LIN {X 0,Y 249.026,Z 523.934,A -85,B 0,C 180,E1 -19032.796,E2 -19032.796} C_VEL
LIN {X 0,Y 250.402,Z 519.579,A -85,B 0,C 180,E1 -19035.438,E2 -19035.438} C_VEL
LIN {X 0,Y 252.113,Z 513.971,A -85,B 0,C 180,E1 -19038.007,E2 -19038.007} C_VEL
LIN {X 0,Y 254.478,Z 506.507,A -85,B 0,C 180,E1 -19040.637,E2 -19040.637} C_VEL
LIN {X 0,Y 257.002,Z 497.79,A -85,B 0,C 180,E1 -19043.014,E2 -19043.014} C_VEL
LIN {X 0,Y 259.635,Z 487.535,A -85,B 0,C 180,E1 -19045.223,E2 -19045.223} C_VEL
LIN {X 0,Y 262.011,Z 477.566,A -85,B 0,C 180,E1 -19046.899,E2 -19046.899} C_VEL
LIN {X 0,Y 264.202,Z 466.893,A -85,B 0,C 180,E1 -19048.33,E2 -19048.33} C_VEL
LIN {X 0,Y 266.285,Z 454.649,A -85,B 0,C 180,E1 -19049.606,E2 -19049.606} C_VEL
LIN {X 0,Y 267.921,Z 441.662,A -85,B 0,C 180,E1 -19050.602,E2 -19050.602} C_VEL
LIN {X 0,Y 269.029,Z 429.527,A -85,B 0,C 180,E1 -19051.238,E2 -19051.238} C_VEL
LIN {X 0,Y 270.232,Z 406.171,A -85,B 0,C 180,E1 -19051.957,E2 -19051.957} C_VEL
LIN {X 0,Y 272.221,Z 363.158,A -85,B 0,C 180,E1 -19053.174,E2 -19053.174} C_VEL
LIN {X 0,Y 265.544,Z 348.107,A -85,B 0,C 180,E1 -19054.833,E2 -19054.833} C_VEL
LIN {X 0,Y 258.825,Z 335.75,A -85,B 0,C 180,E1 -19056.552,E2 -19056.552} C_VEL
LIN {X 0,Y 254.137,Z 328.112,A -85,B 0,C 180,E1 -19057.811,E2 -19057.811} C_VEL
LIN {X 0,Y 251.084,Z 323.594,A -85,B 0,C 180,E1 -19058.661,E2 -19058.661} C_VEL
LIN {X 0,Y 249.464,Z 321.033,A -85,B 0,C 180,E1 -19059.136,E2 -19059.136} C_VEL
LIN {X 0,Y 249.221,Z 320.145,A -85,B 0,C 180,E1 -19059.29,E2 -19059.29} C_VEL
LIN {X 0,Y 249.065,Z 319.467,A -85,B 0,C 180,E1 -19059.777,E2 -19059.777} C_VEL
LIN {X 0,Y 249.159,Z 319.446,A -85,B 0,C 180,E1 -19063.616,E2 -19063.616} C_VEL
LIN {X 0,Y 249.193,Z 319.441,A -85,B 0,C 180,E1 -19068.614,E2 -19068.614} C_VEL
LIN {X 0,Y 249.408,Z 319.413,A -85,B 0,C 180,E1 -19071.9,E2 -19071.9} C_VEL
LIN {X 0,Y 249.252,Z 319.432,A -85,B 0,C 180,E1 -19075.148,E2 -19075.148} C_VEL
LIN {X 0,Y 249.36,Z 319.415,A -85,B 0,C 180,E1 -19076.547,E2 -19076.547} C_VEL
LIN {X 0,Y 249.147,Z 319.448,A -85,B 0,C 180,E1 -19077.45,E2 -19077.45} C_VEL
LIN {X 0,Y 247.894,Z 319.605,A -85,B 0,C 180,E1 -19078.785,E2 -19078.785} C_VEL
LIN {X 0,Y 242.676,Z 320.249,A -85,B 0,C 180,E1 -19082.817,E2 -19082.817} C_VEL
LIN {X 0,Y 242.282,Z 320.293,A -85,B 0,C 180,E1 -19083.759,E2 -19083.759} C_VEL
LIN {X 0,Y 242.387,Z 320.287,A -85,B 0,C 180,E1 -19086.66,E2 -19086.66} C_VEL
LIN {X 0,Y 242.274,Z 320.307,A -85,B 0,C 180,E1 -19090.023,E2 -19090.023} C_VEL
LIN {X 0,Y 242.104,Z 320.321,A -85,B 0,C 180,E1 -19095.145,E2 -19095.145} C_VEL
LIN {X 0,Y 242.049,Z 320.332,A -85,B 0,C 180,E1 -19098.626,E2 -19098.626} C_VEL
LIN {X 0,Y 242.035,Z 320.332,A -85,B 0,C 180,E1 -19102.178,E2 -19102.178} C_VEL
LIN {X 0,Y 242.033,Z 320.33,A -85,B 0,C 180,E1 -19105.842,E2 -19105.842} C_VEL
LIN {X 0,Y 241.997,Z 320.336,A -85,B 0,C 180,E1 -19109.585,E2 -19109.585} C_VEL
LIN {X 0,Y 241.961,Z 320.346,A -85,B 0,C 180,E1 -19113.496,E2 -19113.496} C_VEL
LIN {X 0,Y 242,Z 320.338,A -85,B 0,C 180,E1 -19117.58,E2 -19117.58} C_VEL
LIN {X 0,Y 242.017,Z 320.34,A -85,B 0,C 180,E1 -19121.906,E2 -19121.906} C_VEL
LIN {X 0,Y 242.019,Z 320.432,A -85,B 0,C 180,E1 -19125.685,E2 -19125.685} C_VEL
LIN {X 0,Y 244.031,Z 326.812,A -85,B 0,C 180,E1 -19129.112,E2 -19129.112} C_VEL
LIN {X 0,Y 245.742,Z 332.805,A -85,B 0,C 180,E1 -19132.023,E2 -19132.023} C_VEL
LIN {X 0,Y 248.529,Z 337.73,A -85,B 0,C 180,E1 -19132.878,E2 -19132.878} C_VEL
LIN {X 0,Y 254.858,Z 349.777,A -85,B 0,C 180,E1 -19134.724,E2 -19134.724} C_VEL
LIN {X 0,Y 260.505,Z 361.853,A -85,B 0,C 180,E1 -19136.281,E2 -19136.281} C_VEL
LIN {X 0,Y 262.541,Z 367.254,A -85,B 0,C 180,E1 -19136.855,E2 -19136.855} C_VEL
LIN {X 0,Y 264.938,Z 384.313,A -85,B 0,C 180,E1 -19137.905,E2 -19137.905} C_VEL
LIN {X 0,Y 265.403,Z 390.459,A -85,B 0,C 180,E1 -19138.206,E2 -19138.206} C_VEL
LIN {X 0,Y 262.759,Z 444.06,A -85,B 0,C 180,E1 -19139.798,E2 -19139.798} C_VEL
LIN {X 0,Y 261.252,Z 457.92,A -85,B 0,C 180,E1 -19140.495,E2 -19140.495} C_VEL
LIN {X 0,Y 259.436,Z 469.841,A -85,B 0,C 180,E1 -19141.378,E2 -19141.378} C_VEL
LIN {X 0,Y 257.137,Z 481.502,A -85,B 0,C 180,E1 -19142.542,E2 -19142.542} C_VEL
LIN {X 0,Y 254.668,Z 492.793,A -85,B 0,C 180,E1 -19144.025,E2 -19144.025} C_VEL
LIN {X 0,Y 252.027,Z 503.055,A -85,B 0,C 180,E1 -19145.72,E2 -19145.72} C_VEL
LIN {X 0,Y 249.478,Z 512.316,A -85,B 0,C 180,E1 -19147.655,E2 -19147.655} C_VEL
LIN {X 0,Y 246.894,Z 521.368,A -85,B 0,C 180,E1 -19150.033,E2 -19150.033} C_VEL
LIN {X 0,Y 244.72,Z 528.699,A -85,B 0,C 180,E1 -19152.457,E2 -19152.457} C_VEL
LIN {X 0,Y 242.867,Z 534.602,A -85,B 0,C 180,E1 -19154.911,E2 -19154.911} C_VEL
LIN {X 0,Y 241.478,Z 539.276,A -85,B 0,C 180,E1 -19157.398,E2 -19157.398} C_VEL
LIN {X 0,Y 240.6,Z 542.861,A -85,B 0,C 180,E1 -19159.912,E2 -19159.912} C_VEL
LIN {X 0,Y 240.202,Z 544.688,A -85,B 0,C 180,E1 -19161.594,E2 -19161.594} C_VEL
LIN {X 0,Y 239.799,Z 547.099,A -85,B 0,C 180,E1 -19164.962,E2 -19164.962} C_VEL
LIN {X 0,Y 239.799,Z 547.72,A -85,B 0,C 180,E1 -19166.645,E2 -19166.645} C_VEL
LIN {X 0,Y 239.903,Z 547.911,A -85,B 0,C 180,E1 -19168.327,E2 -19168.327} C_VEL
LIN {X 0,Y 239.958,Z 547.686,A -85,B 0,C 180,E1 -19170.005,E2 -19170.005} C_VEL
LIN {X 0,Y 239.917,Z 547.061,A -85,B 0,C 180,E1 -19171.684,E2 -19171.684} C_VEL
LIN {X 0,Y 239.841,Z 546.03,A -85,B 0,C 180,E1 -19173.365,E2 -19173.365} C_VEL
LIN {X 0,Y 239.849,Z 544.537,A -85,B 0,C 180,E1 -19175.048,E2 -19175.048} C_VEL
LIN {X 0,Y 240.047,Z 541.476,A -85,B 0,C 180,E1 -19177.576,E2 -19177.576} C_VEL
LIN {X 0,Y 240.503,Z 537.321,A -85,B 0,C 180,E1 -19180.103,E2 -19180.103} C_VEL
LIN {X 0,Y 241.444,Z 530.931,A -85,B 0,C 180,E1 -19183.042,E2 -19183.042} C_VEL
LIN {X 0,Y 242.804,Z 523.965,A -85,B 0,C 180,E1 -19185.535,E2 -19185.535} C_VEL
LIN {X 0,Y 244.46,Z 515.208,A -85,B 0,C 180,E1 -19188.006,E2 -19188.006} C_VEL
LIN {X 0,Y 246.228,Z 505.21,A -85,B 0,C 180,E1 -19190.252,E2 -19190.252} C_VEL
LIN {X 0,Y 248.095,Z 495.105,A -85,B 0,C 180,E1 -19192.05,E2 -19192.05} C_VEL
LIN {X 0,Y 249.963,Z 483.875,A -85,B 0,C 180,E1 -19193.623,E2 -19193.623} C_VEL
LIN {X 0,Y 251.793,Z 471.326,A -85,B 0,C 180,E1 -19194.975,E2 -19194.975} C_VEL
LIN {X 0,Y 253.237,Z 458.517,A -85,B 0,C 180,E1 -19195.978,E2 -19195.978} C_VEL
LIN {X 0,Y 254.374,Z 445.256,A -85,B 0,C 180,E1 -19196.674,E2 -19196.674} C_VEL
LIN {X 0,Y 256.515,Z 387.54,A -85,B 0,C 180,E1 -19198.405,E2 -19198.405} C_VEL
LIN {X 0,Y 252.725,Z 358.428,A -85,B 0,C 180,E1 -19199.754,E2 -19199.754} C_VEL
LIN {X 0,Y 251.517,Z 351.799,A -85,B 0,C 180,E1 -19200.103,E2 -19200.103} C_VEL
LIN {X 0,Y 245.361,Z 335.617,A -85,B 0,C 180,E1 -19201.356,E2 -19201.356} C_VEL
LIN {X 0,Y 243.532,Z 326.882,A -85,B 0,C 180,E1 -19204.762,E2 -19204.762} C_VEL
LIN {X 0,Y 242.052,Z 320.333,A -85,B 0,C 180,E1 -19207.459,E2 -19207.459} C_VEL
LIN {X 0,Y 241.941,Z 320.35,A -85,B 0,C 180,E1 -19211.925,E2 -19211.925} C_VEL
LIN {X 0,Y 241.933,Z 320.352,A -85,B 0,C 180,E1 -19216.575,E2 -19216.575} C_VEL
LIN {X 0,Y 242.001,Z 320.339,A -85,B 0,C 180,E1 -19221.642,E2 -19221.642} C_VEL
LIN {X 0,Y 241.986,Z 320.343,A -85,B 0,C 180,E1 -19224.489,E2 -19224.489} C_VEL
LIN {X 0,Y 241.975,Z 320.346,A -85,B 0,C 180,E1 -19228.48,E2 -19228.48} C_VEL
LIN {X 0,Y 242.006,Z 320.34,A -85,B 0,C 180,E1 -19232.312,E2 -19232.312} C_VEL
LIN {X 0,Y 242.044,Z 320.331,A -85,B 0,C 180,E1 -19236.015,E2 -19236.015} C_VEL
LIN {X 0,Y 241.998,Z 320.336,A -85,B 0,C 180,E1 -19239.604,E2 -19239.604} C_VEL
LIN {X 0,Y 242.12,Z 320.304,A -85,B 0,C 180,E1 -19243.319,E2 -19243.319} C_VEL
LIN {X 0,Y 242.168,Z 320.315,A -85,B 0,C 180,E1 -19248.279,E2 -19248.279} C_VEL
LIN {X 0,Y 242.399,Z 320.288,A -85,B 0,C 180,E1 -19251.665,E2 -19251.665} C_VEL
LIN {X 0,Y 242.423,Z 320.281,A -85,B 0,C 180,E1 -19253.341,E2 -19253.341} C_VEL
LIN {X 0,Y 242.636,Z 320.233,A -85,B 0,C 180,E1 -19258.34,E2 -19258.34} C_VEL
LIN {X 0,Y 242.634,Z 320.251,A -85,B 0,C 180,E1 -19261.66,E2 -19261.66} C_VEL
LIN {X 0,Y 242.395,Z 320.289,A -85,B 0,C 180,E1 -19266.66,E2 -19266.66} C_VEL
LIN {X 0,Y 242.266,Z 320.3,A -85,B 0,C 180,E1 -19270.024,E2 -19270.024} C_VEL
LIN {X 0,Y 242.126,Z 320.323,A -85,B 0,C 180,E1 -19275.144,E2 -19275.144} C_VEL
LIN {X 0,Y 242.026,Z 320.326,A -85,B 0,C 180,E1 -19278.628,E2 -19278.628} C_VEL
LIN {X 0,Y 241.978,Z 320.343,A -85,B 0,C 180,E1 -19282.183,E2 -19282.183} C_VEL
LIN {X 0,Y 241.992,Z 320.339,A -85,B 0,C 180,E1 -19285.826,E2 -19285.826} C_VEL
LIN {X 0,Y 241.967,Z 320.324,A -85,B 0,C 180,E1 -19289.589,E2 -19289.589} C_VEL
LIN {X 0,Y 241.973,Z 320.324,A -85,B 0,C 180,E1 -19293.494,E2 -19293.494} C_VEL
LIN {X 0,Y 241.971,Z 320.34,A -85,B 0,C 180,E1 -19297.585,E2 -19297.585} C_VEL
LIN {X 0,Y 241.905,Z 320.348,A -85,B 0,C 180,E1 -19301.93,E2 -19301.93} C_VEL
LIN {X 0,Y 241.891,Z 320.356,A -85,B 0,C 180,E1 -19306.582,E2 -19306.582} C_VEL
LIN {X 0,Y 241.936,Z 320.343,A -85,B 0,C 180,E1 -19310.273,E2 -19310.273} C_VEL
LIN {X 0,Y 241.981,Z 320.343,A -85,B 0,C 180,E1 -19314.484,E2 -19314.484} C_VEL
LIN {X 0,Y 241.937,Z 320.35,A -85,B 0,C 180,E1 -19318.47,E2 -19318.47} C_VEL
LIN {X 0,Y 241.968,Z 320.344,A -85,B 0,C 180,E1 -19322.304,E2 -19322.304} C_VEL
LIN {X 0,Y 242.03,Z 320.334,A -85,B 0,C 180,E1 -19326.009,E2 -19326.009} C_VEL
LIN {X 0,Y 242,Z 320.341,A -85,B 0,C 180,E1 -19329.6,E2 -19329.6} C_VEL
LIN {X 0,Y 242.122,Z 320.327,A -85,B 0,C 180,E1 -19333.312,E2 -19333.312} C_VEL
LIN {X 0,Y 242.173,Z 320.316,A -85,B 0,C 180,E1 -19338.274,E2 -19338.274} C_VEL
LIN {X 0,Y 242.376,Z 320.29,A -85,B 0,C 180,E1 -19341.659,E2 -19341.659} C_VEL
LIN {X 0,Y 242.4,Z 320.291,A -85,B 0,C 180,E1 -19343.335,E2 -19343.335} C_VEL
LIN {X 0,Y 242.622,Z 320.26,A -85,B 0,C 180,E1 -19348.335,E2 -19348.335} C_VEL
LIN {X 0,Y 242.638,Z 320.438,A -85,B 0,C 180,E1 -19350.461,E2 -19350.461} C_VEL
LIN {X 0,Y 243.698,Z 323.226,A -85,B 0,C 180,E1 -19350.686,E2 -19350.686} C_VEL
LIN {X 0,Y 247.603,Z 332.184,A -85,B 0,C 180,E1 -19351.45,E2 -19351.45} C_VEL
LIN {X 0,Y 254.32,Z 349.239,A -85,B 0,C 180,E1 -19352.752,E2 -19352.752} C_VEL
LIN {X 0,Y 257.363,Z 357.984,A -85,B 0,C 180,E1 -19353.352,E2 -19353.352} C_VEL
LIN {X 0,Y 254.717,Z 426.897,A -85,B 0,C 180,E1 -19355.391,E2 -19355.391} C_VEL
LIN {X 0,Y 253.733,Z 440.855,A -85,B 0,C 180,E1 -19356.14,E2 -19356.14} C_VEL
LIN {X 0,Y 252.489,Z 453.86,A -85,B 0,C 180,E1 -19357.19,E2 -19357.19} C_VEL
LIN {X 0,Y 250.977,Z 465.457,A -85,B 0,C 180,E1 -19358.448,E2 -19358.448} C_VEL
LIN {X 0,Y 249.262,Z 476.237,A -85,B 0,C 180,E1 -19359.939,E2 -19359.939} C_VEL
LIN {X 0,Y 247.528,Z 486.205,A -85,B 0,C 180,E1 -19361.665,E2 -19361.665} C_VEL
LIN {X 0,Y 245.738,Z 495.959,A -85,B 0,C 180,E1 -19363.791,E2 -19363.791} C_VEL
LIN {X 0,Y 243.947,Z 505.16,A -85,B 0,C 180,E1 -19366.307,E2 -19366.307} C_VEL
LIN {X 0,Y 242.666,Z 511.758,A -85,B 0,C 180,E1 -19368.57,E2 -19368.57} C_VEL
LIN {X 0,Y 241.472,Z 518.139,A -85,B 0,C 180,E1 -19371.352,E2 -19371.352} C_VEL
LIN {X 0,Y 240.693,Z 522.973,A -85,B 0,C 180,E1 -19374.121,E2 -19374.121} C_VEL
LIN {X 0,Y 240.213,Z 525.551,A -85,B 0,C 180,E1 -19376.023,E2 -19376.023} C_VEL
LIN {X 0,Y 239.738,Z 527.941,A -85,B 0,C 180,E1 -19378.422,E2 -19378.422} C_VEL
LIN {X 0,Y 239.585,Z 528.991,A -85,B 0,C 180,E1 -19379.904,E2 -19379.904} C_VEL
LIN {X 0,Y 239.562,Z 529.858,A -85,B 0,C 180,E1 -19381.866,E2 -19381.866} C_VEL
LIN {X 0,Y 239.738,Z 530.179,A -85,B 0,C 180,E1 -19384.832,E2 -19384.832} C_VEL
LIN {X 0,Y 240.236,Z 529.227,A -85,B 0,C 180,E1 -19387.894,E2 -19387.894} C_VEL
LIN {X 0,Y 241.105,Z 527.123,A -85,B 0,C 180,E1 -19390.722,E2 -19390.722} C_VEL
LIN {X 0,Y 242.246,Z 523.843,A -85,B 0,C 180,E1 -19393.506,E2 -19393.506} C_VEL
LIN {X 0,Y 243.754,Z 519.379,A -85,B 0,C 180,E1 -19396.213,E2 -19396.213} C_VEL
LIN {X 0,Y 245.683,Z 513.607,A -85,B 0,C 180,E1 -19398.857,E2 -19398.857} C_VEL
LIN {X 0,Y 248.116,Z 506.269,A -85,B 0,C 180,E1 -19401.452,E2 -19401.452} C_VEL
LIN {X 0,Y 250.841,Z 497.136,A -85,B 0,C 180,E1 -19403.958,E2 -19403.958} C_VEL
LIN {X 0,Y 253.34,Z 487.96,A -85,B 0,C 180,E1 -19405.958,E2 -19405.958} C_VEL
LIN {X 0,Y 255.802,Z 478.185,A -85,B 0,C 180,E1 -19407.65,E2 -19407.65} C_VEL
LIN {X 0,Y 258.155,Z 467.333,A -85,B 0,C 180,E1 -19409.136,E2 -19409.136} C_VEL
LIN {X 0,Y 260.397,Z 454.641,A -85,B 0,C 180,E1 -19410.483,E2 -19410.483} C_VEL
LIN {X 0,Y 262.048,Z 442.095,A -85,B 0,C 180,E1 -19411.458,E2 -19411.458} C_VEL
LIN {X 0,Y 263.222,Z 429.745,A -85,B 0,C 180,E1 -19412.116,E2 -19412.116} C_VEL
LIN {X 0,Y 264.502,Z 405.907,A -85,B 0,C 180,E1 -19412.86,E2 -19412.86} C_VEL
LIN {X 0,Y 266.484,Z 365.311,A -85,B 0,C 180,E1 -19414.027,E2 -19414.027} C_VEL
LIN {X 0,Y 260.565,Z 351.905,A -85,B 0,C 180,E1 -19415.587,E2 -19415.587} C_VEL
LIN {X 0,Y 254.402,Z 340.316,A -85,B 0,C 180,E1 -19417.247,E2 -19417.247} C_VEL
LIN {X 0,Y 249.596,Z 332.463,A -85,B 0,C 180,E1 -19418.604,E2 -19418.604} C_VEL
LIN {X 0,Y 247.303,Z 329.005,A -85,B 0,C 180,E1 -19419.274,E2 -19419.274} C_VEL
LIN {X 0,Y 245.279,Z 325.831,A -85,B 0,C 180,E1 -19419.889,E2 -19419.889} C_VEL
LIN {X 0,Y 242.726,Z 322.681,A -85,B 0,C 180,E1 -19420.66,E2 -19420.66} C_VEL
LIN {X 0,Y 242.084,Z 320.672,A -85,B 0,C 180,E1 -19420.937,E2 -19420.937} C_VEL
LIN {X 0,Y 242.029,Z 320.337,A -85,B 0,C 180,E1 -19421.372,E2 -19421.372} C_VEL
LIN {X 0,Y 242.102,Z 320.329,A -85,B 0,C 180,E1 -19424.855,E2 -19424.855} C_VEL
LIN {X 0,Y 242.275,Z 320.303,A -85,B 0,C 180,E1 -19430.443,E2 -19430.443} C_VEL
LIN {X 0,Y 242.379,Z 320.288,A -85,B 0,C 180,E1 -19433.34,E2 -19433.34} C_VEL
LIN {X 0,Y 242.594,Z 320.265,A -85,B 0,C 180,E1 -19438.34,E2 -19438.34} C_VEL
LIN {X 0,Y 242.594,Z 320.266,A -85,B 0,C 180,E1 -19441.66,E2 -19441.66} C_VEL
LIN {X 0,Y 242.282,Z 320.293,A -85,B 0,C 180,E1 -19443.759,E2 -19443.759} C_VEL
LIN {X 0,Y 241.536,Z 320.395,A -85,B 0,C 180,E1 -19445.148,E2 -19445.148} C_VEL
LIN {X 0,Y 238.687,Z 320.752,A -85,B 0,C 180,E1 -19447.415,E2 -19447.415} C_VEL
LIN {X 0,Y 235.469,Z 321.155,A -85,B 0,C 180,E1 -19450.211,E2 -19450.211} C_VEL
LIN {X 0,Y 235.112,Z 321.189,A -85,B 0,C 180,E1 -19451.179,E2 -19451.179} C_VEL
LIN {X 0,Y 235.058,Z 321.194,A -85,B 0,C 180,E1 -19455.61,E2 -19455.61} C_VEL
LIN {X 0,Y 234.994,Z 321.205,A -85,B 0,C 180,E1 -19459.207,E2 -19459.207} C_VEL
LIN {X 0,Y 234.963,Z 321.212,A -85,B 0,C 180,E1 -19462.883,E2 -19462.883} C_VEL
LIN {X 0,Y 234.936,Z 321.218,A -85,B 0,C 180,E1 -19466.662,E2 -19466.662} C_VEL
LIN {X 0,Y 234.899,Z 321.223,A -85,B 0,C 180,E1 -19470.572,E2 -19470.572} C_VEL
LIN {X 0,Y 234.931,Z 321.216,A -85,B 0,C 180,E1 -19474.638,E2 -19474.638} C_VEL
LIN {X 0,Y 234.971,Z 321.213,A -85,B 0,C 180,E1 -19478.967,E2 -19478.967} C_VEL
LIN {X 0,Y 234.972,Z 321.218,A -85,B 0,C 180,E1 -19483.467,E2 -19483.467} C_VEL
LIN {X 0,Y 234.962,Z 321.348,A -85,B 0,C 180,E1 -19484.064,E2 -19484.064} C_VEL
LIN {X 0,Y 237.368,Z 328.906,A -85,B 0,C 180,E1 -19488.388,E2 -19488.388} C_VEL
LIN {X 0,Y 238.399,Z 332.499,A -85,B 0,C 180,E1 -19490.185,E2 -19490.185} C_VEL
LIN {X 0,Y 241.186,Z 337.207,A -85,B 0,C 180,E1 -19491.131,E2 -19491.131} C_VEL
LIN {X 0,Y 245.517,Z 344.826,A -85,B 0,C 180,E1 -19492.512,E2 -19492.512} C_VEL
LIN {X 0,Y 251.337,Z 356.174,A -85,B 0,C 180,E1 -19494.275,E2 -19494.275} C_VEL
LIN {X 0,Y 257.128,Z 369.32,A -85,B 0,C 180,E1 -19495.947,E2 -19495.947} C_VEL
LIN {X 0,Y 259.348,Z 385.503,A -85,B 0,C 180,E1 -19496.986,E2 -19496.986} C_VEL
LIN {X 0,Y 259.804,Z 390.388,A -85,B 0,C 180,E1 -19497.255,E2 -19497.255} C_VEL
LIN {X 0,Y 257.015,Z 443.859,A -85,B 0,C 180,E1 -19498.878,E2 -19498.878} C_VEL
LIN {X 0,Y 255.445,Z 457.689,A -85,B 0,C 180,E1 -19499.583,E2 -19499.583} C_VEL
LIN {X 0,Y 253.465,Z 470.082,A -85,B 0,C 180,E1 -19500.525,E2 -19500.525} C_VEL
LIN {X 0,Y 250.919,Z 482.419,A -85,B 0,C 180,E1 -19501.802,E2 -19501.802} C_VEL
LIN {X 0,Y 248.352,Z 493.499,A -85,B 0,C 180,E1 -19503.313,E2 -19503.313} C_VEL
LIN {X 0,Y 245.597,Z 503.552,A -85,B 0,C 180,E1 -19505.041,E2 -19505.041} C_VEL
LIN {X 0,Y 242.946,Z 512.668,A -85,B 0,C 180,E1 -19507.02,E2 -19507.02} C_VEL
LIN {X 0,Y 240.217,Z 521.595,A -85,B 0,C 180,E1 -19509.454,E2 -19509.454} C_VEL
LIN {X 0,Y 237.933,Z 528.817,A -85,B 0,C 180,E1 -19511.939,E2 -19511.939} C_VEL
LIN {X 0,Y 235.986,Z 534.622,A -85,B 0,C 180,E1 -19514.46,E2 -19514.46} C_VEL
LIN {X 0,Y 234.519,Z 539.231,A -85,B 0,C 180,E1 -19517.018,E2 -19517.018} C_VEL
LIN {X 0,Y 233.572,Z 542.765,A -85,B 0,C 180,E1 -19519.606,E2 -19519.606} C_VEL
LIN {X 0,Y 233.17,Z 544.545,A -85,B 0,C 180,E1 -19521.338,E2 -19521.338} C_VEL
LIN {X 0,Y 232.728,Z 546.901,A -85,B 0,C 180,E1 -19524.808,E2 -19524.808} C_VEL
LIN {X 0,Y 232.704,Z 547.482,A -85,B 0,C 180,E1 -19526.543,E2 -19526.543} C_VEL
LIN {X 0,Y 232.81,Z 547.63,A -85,B 0,C 180,E1 -19528.276,E2 -19528.276} C_VEL
LIN {X 0,Y 232.888,Z 547.38,A -85,B 0,C 180,E1 -19530.006,E2 -19530.006} C_VEL
LIN {X 0,Y 232.825,Z 546.728,A -85,B 0,C 180,E1 -19531.735,E2 -19531.735} C_VEL
LIN {X 0,Y 232.767,Z 544.462,A -85,B 0,C 180,E1 -19534.875,E2 -19534.875} C_VEL
LIN {X 0,Y 233.001,Z 541.005,A -85,B 0,C 180,E1 -19537.806,E2 -19537.806} C_VEL
LIN {X 0,Y 233.482,Z 536.786,A -85,B 0,C 180,E1 -19540.41,E2 -19540.41} C_VEL
LIN {X 0,Y 234.502,Z 530.329,A -85,B 0,C 180,E1 -19543.435,E2 -19543.435} C_VEL
LIN {X 0,Y 235.887,Z 523.268,A -85,B 0,C 180,E1 -19546.002,E2 -19546.002} C_VEL
LIN {X 0,Y 237.533,Z 514.944,A -85,B 0,C 180,E1 -19548.4,E2 -19548.4} C_VEL
LIN {X 0,Y 239.343,Z 505.269,A -85,B 0,C 180,E1 -19550.636,E2 -19550.636} C_VEL
LIN {X 0,Y 241.259,Z 495.249,A -85,B 0,C 180,E1 -19552.483,E2 -19552.483} C_VEL
LIN {X 0,Y 243.177,Z 484.12,A -85,B 0,C 180,E1 -19554.097,E2 -19554.097} C_VEL
LIN {X 0,Y 245.041,Z 471.695,A -85,B 0,C 180,E1 -19555.485,E2 -19555.485} C_VEL
LIN {X 0,Y 246.505,Z 459.954,A -85,B 0,C 180,E1 -19556.458,E2 -19556.458} C_VEL
LIN {X 0,Y 247.657,Z 446.77,A -85,B 0,C 180,E1 -19557.21,E2 -19557.21} C_VEL
LIN {X 0,Y 248.591,Z 425.841,A -85,B 0,C 180,E1 -19557.908,E2 -19557.908} C_VEL
LIN {X 0,Y 249.931,Z 387.258,A -85,B 0,C 180,E1 -19559.071,E2 -19559.071} C_VEL
LIN {X 0,Y 245.978,Z 357.308,A -85,B 0,C 180,E1 -19560.508,E2 -19560.508} C_VEL
LIN {X 0,Y 245.065,Z 353.574,A -85,B 0,C 180,E1 -19560.739,E2 -19560.739} C_VEL
LIN {X 0,Y 238.12,Z 335.305,A -85,B 0,C 180,E1 -19562.234,E2 -19562.234} C_VEL
LIN {X 0,Y 235.775,Z 324.601,A -85,B 0,C 180,E1 -19566.599,E2 -19566.599} C_VEL
LIN {X 0,Y 234.96,Z 321.22,A -85,B 0,C 180,E1 -19568.096,E2 -19568.096} C_VEL
LIN {X 0,Y 234.888,Z 321.231,A -85,B 0,C 180,E1 -19571.581,E2 -19571.581} C_VEL
LIN {X 0,Y 234.891,Z 321.229,A -85,B 0,C 180,E1 -19575.9,E2 -19575.9} C_VEL
LIN {X 0,Y 234.88,Z 321.227,A -85,B 0,C 180,E1 -19578.831,E2 -19578.831} C_VEL
LIN {X 0,Y 234.923,Z 321.222,A -85,B 0,C 180,E1 -19583.25,E2 -19583.25} C_VEL
LIN {X 0,Y 234.96,Z 321.218,A -85,B 0,C 180,E1 -19587.425,E2 -19587.425} C_VEL
LIN {X 0,Y 234.942,Z 321.22,A -85,B 0,C 180,E1 -19591.405,E2 -19591.405} C_VEL
LIN {X 0,Y 234.983,Z 321.212,A -85,B 0,C 180,E1 -19595.246,E2 -19595.246} C_VEL
LIN {X 0,Y 234.95,Z 321.218,A -85,B 0,C 180,E1 -19598.964,E2 -19598.964} C_VEL
LIN {X 0,Y 235.062,Z 321.183,A -85,B 0,C 180,E1 -19603.094,E2 -19603.094} C_VEL
LIN {X 0,Y 235.1,Z 321.196,A -85,B 0,C 180,E1 -19607.921,E2 -19607.921} C_VEL
LIN {X 0,Y 235.328,Z 321.17,A -85,B 0,C 180,E1 -19611.412,E2 -19611.412} C_VEL
LIN {X 0,Y 235.373,Z 321.161,A -85,B 0,C 180,E1 -19613.14,E2 -19613.14} C_VEL
LIN {X 0,Y 235.595,Z 321.108,A -85,B 0,C 180,E1 -19618.291,E2 -19618.291} C_VEL
LIN {X 0,Y 235.594,Z 321.128,A -85,B 0,C 180,E1 -19621.709,E2 -19621.709} C_VEL
LIN {X 0,Y 235.345,Z 321.167,A -85,B 0,C 180,E1 -19626.86,E2 -19626.86} C_VEL
LIN {X 0,Y 235.191,Z 321.18,A -85,B 0,C 180,E1 -19630.329,E2 -19630.329} C_VEL
LIN {X 0,Y 235.075,Z 321.203,A -85,B 0,C 180,E1 -19635.609,E2 -19635.609} C_VEL
LIN {X 0,Y 234.967,Z 321.205,A -85,B 0,C 180,E1 -19639.209,E2 -19639.209} C_VEL
LIN {X 0,Y 234.921,Z 321.219,A -85,B 0,C 180,E1 -19642.887,E2 -19642.887} C_VEL
LIN {X 0,Y 234.91,Z 321.214,A -85,B 0,C 180,E1 -19646.665,E2 -19646.665} C_VEL
LIN {X 0,Y 234.891,Z 321.193,A -85,B 0,C 180,E1 -19650.574,E2 -19650.574} C_VEL
LIN {X 0,Y 234.905,Z 321.212,A -85,B 0,C 180,E1 -19654.643,E2 -19654.643} C_VEL
LIN {X 0,Y 234.92,Z 321.221,A -85,B 0,C 180,E1 -19658.934,E2 -19658.934} C_VEL
LIN {X 0,Y 234.86,Z 321.225,A -85,B 0,C 180,E1 -19664.092,E2 -19664.092} C_VEL
LIN {X 0,Y 234.852,Z 321.226,A -85,B 0,C 180,E1 -19668.821,E2 -19668.821} C_VEL
LIN {X 0,Y 234.926,Z 321.222,A -85,B 0,C 180,E1 -19671.076,E2 -19671.076} C_VEL
LIN {X 0,Y 234.905,Z 321.22,A -85,B 0,C 180,E1 -19675.354,E2 -19675.354} C_VEL
LIN {X 0,Y 234.894,Z 321.226,A -85,B 0,C 180,E1 -19679.423,E2 -19679.423} C_VEL
LIN {X 0,Y 234.976,Z 321.217,A -85,B 0,C 180,E1 -19683.804,E2 -19683.804} C_VEL
LIN {X 0,Y 234.973,Z 321.218,A -85,B 0,C 180,E1 -19688.004,E2 -19688.004} C_VEL
LIN {X 0,Y 235.063,Z 321.209,A -85,B 0,C 180,E1 -19693.088,E2 -19693.088} C_VEL
LIN {X 0,Y 235.104,Z 321.197,A -85,B 0,C 180,E1 -19697.917,E2 -19697.917} C_VEL
LIN {X 0,Y 235.316,Z 321.169,A -85,B 0,C 180,E1 -19701.407,E2 -19701.407} C_VEL
LIN {X 0,Y 235.352,Z 321.168,A -85,B 0,C 180,E1 -19703.135,E2 -19703.135} C_VEL
LIN {X 0,Y 235.58,Z 321.137,A -85,B 0,C 180,E1 -19708.285,E2 -19708.285} C_VEL
LIN {X 0,Y 235.584,Z 321.142,A -85,B 0,C 180,E1 -19709.621,E2 -19709.621} C_VEL
LIN {X 0,Y 236.502,Z 323.833,A -85,B 0,C 180,E1 -19709.835,E2 -19709.835} C_VEL
LIN {X 0,Y 240.954,Z 333.301,A -85,B 0,C 180,E1 -19710.72,E2 -19710.72} C_VEL
LIN {X 0,Y 248.512,Z 352.797,A -85,B 0,C 180,E1 -19712.259,E2 -19712.259} C_VEL
LIN {X 0,Y 250.863,Z 360.046,A -85,B 0,C 180,E1 -19712.754,E2 -19712.754} C_VEL
LIN {X 0,Y 248.133,Z 427.294,A -85,B 0,C 180,E1 -19714.792,E2 -19714.792} C_VEL
LIN {X 0,Y 247.136,Z 440.947,A -85,B 0,C 180,E1 -19715.542,E2 -19715.542} C_VEL
LIN {X 0,Y 245.909,Z 453.423,A -85,B 0,C 180,E1 -19716.559,E2 -19716.559} C_VEL
LIN {X 0,Y 244.353,Z 465.146,A -85,B 0,C 180,E1 -19717.846,E2 -19717.846} C_VEL
LIN {X 0,Y 242.514,Z 476.378,A -85,B 0,C 180,E1 -19719.428,E2 -19719.428} C_VEL
LIN {X 0,Y 240.533,Z 487.213,A -85,B 0,C 180,E1 -19721.368,E2 -19721.368} C_VEL
LIN {X 0,Y 238.674,Z 497.228,A -85,B 0,C 180,E1 -19723.658,E2 -19723.658} C_VEL
LIN {X 0,Y 237.028,Z 505.179,A -85,B 0,C 180,E1 -19725.911,E2 -19725.911} C_VEL
LIN {X 0,Y 235.658,Z 512.068,A -85,B 0,C 180,E1 -19728.333,E2 -19728.333} C_VEL
LIN {X 0,Y 234.454,Z 518.205,A -85,B 0,C 180,E1 -19731.075,E2 -19731.075} C_VEL
LIN {X 0,Y 233.651,Z 523.118,A -85,B 0,C 180,E1 -19733.95,E2 -19733.95} C_VEL
LIN {X 0,Y 232.895,Z 526.79,A -85,B 0,C 180,E1 -19736.906,E2 -19736.906} C_VEL
LIN {X 0,Y 232.597,Z 528.531,A -85,B 0,C 180,E1 -19738.902,E2 -19738.902} C_VEL
LIN {X 0,Y 232.461,Z 530.174,A -85,B 0,C 180,E1 -19742.164,E2 -19742.164} C_VEL
LIN {X 0,Y 232.692,Z 530.432,A -85,B 0,C 180,E1 -19745.365,E2 -19745.365} C_VEL
LIN {X 0,Y 233.279,Z 529.383,A -85,B 0,C 180,E1 -19748.436,E2 -19748.436} C_VEL
LIN {X 0,Y 234.251,Z 527.123,A -85,B 0,C 180,E1 -19751.405,E2 -19751.405} C_VEL
LIN {X 0,Y 235.499,Z 523.75,A -85,B 0,C 180,E1 -19754.255,E2 -19754.255} C_VEL
LIN {X 0,Y 237.162,Z 519.183,A -85,B 0,C 180,E1 -19757.033,E2 -19757.033} C_VEL
LIN {X 0,Y 239.3,Z 513.24,A -85,B 0,C 180,E1 -19759.769,E2 -19759.769} C_VEL
LIN {X 0,Y 241.874,Z 505.792,A -85,B 0,C 180,E1 -19762.397,E2 -19762.397} C_VEL
LIN {X 0,Y 244.481,Z 497.537,A -85,B 0,C 180,E1 -19764.695,E2 -19764.695} C_VEL
LIN {X 0,Y 247.022,Z 488.674,A -85,B 0,C 180,E1 -19766.678,E2 -19766.678} C_VEL
LIN {X 0,Y 249.581,Z 479.074,A -85,B 0,C 180,E1 -19768.393,E2 -19768.393} C_VEL
LIN {X 0,Y 252.243,Z 467.298,A -85,B 0,C 180,E1 -19770.042,E2 -19770.042} C_VEL
LIN {X 0,Y 254.524,Z 454.918,A -85,B 0,C 180,E1 -19771.372,E2 -19771.372} C_VEL
LIN {X 0,Y 256.266,Z 442.397,A -85,B 0,C 180,E1 -19772.361,E2 -19772.361} C_VEL
LIN {X 0,Y 257.444,Z 430.603,A -85,B 0,C 180,E1 -19773.01,E2 -19773.01} C_VEL
LIN {X 0,Y 258.615,Z 410.729,A -85,B 0,C 180,E1 -19773.662,E2 -19773.662} C_VEL
LIN {X 0,Y 260.787,Z 367.352,A -85,B 0,C 180,E1 -19774.947,E2 -19774.947} C_VEL
LIN {X 0,Y 255.671,Z 355.747,A -85,B 0,C 180,E1 -19776.361,E2 -19776.361} C_VEL
LIN {X 0,Y 249.838,Z 344.615,A -85,B 0,C 180,E1 -19778.026,E2 -19778.026} C_VEL
LIN {X 0,Y 244.951,Z 336.58,A -85,B 0,C 180,E1 -19779.477,E2 -19779.477} C_VEL
LIN {X 0,Y 240.811,Z 330.383,A -85,B 0,C 180,E1 -19780.777,E2 -19780.777} C_VEL
LIN {X 0,Y 238.564,Z 327.157,A -85,B 0,C 180,E1 -19781.52,E2 -19781.52} C_VEL
LIN {X 0,Y 238,Z 326.175,A -85,B 0,C 180,E1 -19781.72,E2 -19781.72} C_VEL
LIN {X 0,Y 235.951,Z 323.972,A -85,B 0,C 180,E1 -19782.39,E2 -19782.39} C_VEL
LIN {X 0,Y 235.038,Z 321.21,A -85,B 0,C 180,E1 -19782.823,E2 -19782.823} C_VEL
LIN {X 0,Y 235.043,Z 321.203,A -85,B 0,C 180,E1 -19786.16,E2 -19786.16} C_VEL
LIN {X 0,Y 235.283,Z 321.177,A -85,B 0,C 180,E1 -19791.411,E2 -19791.411} C_VEL
LIN {X 0,Y 235.329,Z 321.164,A -85,B 0,C 180,E1 -19793.139,E2 -19793.139} C_VEL
LIN {X 0,Y 235.553,Z 321.142,A -85,B 0,C 180,E1 -19798.29,E2 -19798.29} C_VEL
LIN {X 0,Y 235.554,Z 321.142,A -85,B 0,C 180,E1 -19801.71,E2 -19801.71} C_VEL
LIN {X 0,Y 235.338,Z 321.162,A -85,B 0,C 180,E1 -19806.861,E2 -19806.861} C_VEL
LIN {X 0,Y 235.199,Z 321.188,A -85,B 0,C 180,E1 -19810.328,E2 -19810.328} C_VEL
LIN {X 0,Y 235.112,Z 321.189,A -85,B 0,C 180,E1 -19811.179,E2 -19811.179} C_VEL
LIN {X 0,Y 234.376,Z 321.279,A -85,B 0,C 180,E1 -19812.609,E2 -19812.609} C_VEL
LIN {X 0,Y 231.488,Z 321.645,A -85,B 0,C 180,E1 -19814.942,E2 -19814.942} C_VEL
LIN {X 0,Y 229.064,Z 321.947,A -85,B 0,C 180,E1 -19816.844,E2 -19816.844} C_VEL
LIN {X 0,Y 228.016,Z 322.079,A -85,B 0,C 180,E1 -19818.32,E2 -19818.32} C_VEL
LIN {X 0,Y 227.923,Z 322.081,A -85,B 0,C 180,E1 -19818.821,E2 -19818.821} C_VEL
LIN {X 0,Y 227.943,Z 322.087,A -85,B 0,C 180,E1 -19822.361,E2 -19822.361} C_VEL
LIN {X 0,Y 227.91,Z 322.093,A -85,B 0,C 180,E1 -19826.606,E2 -19826.606} C_VEL
LIN {X 0,Y 227.876,Z 322.099,A -85,B 0,C 180,E1 -19830.3,E2 -19830.3} C_VEL
LIN {X 0,Y 227.86,Z 322.103,A -85,B 0,C 180,E1 -19833.723,E2 -19833.723} C_VEL
LIN {X 0,Y 227.865,Z 322.096,A -85,B 0,C 180,E1 -19838.087,E2 -19838.087} C_VEL
LIN {X 0,Y 227.929,Z 322.208,A -85,B 0,C 180,E1 -19842.206,E2 -19842.206} C_VEL
LIN {X 0,Y 230.452,Z 329.982,A -85,B 0,C 180,E1 -19847.048,E2 -19847.048} C_VEL
LIN {X 0,Y 231.104,Z 332.064,A -85,B 0,C 180,E1 -19848.132,E2 -19848.132} C_VEL
LIN {X 0,Y 234.181,Z 337.127,A -85,B 0,C 180,E1 -19849.275,E2 -19849.275} C_VEL
LIN {X 0,Y 238.966,Z 345.21,A -85,B 0,C 180,E1 -19850.953,E2 -19850.953} C_VEL
LIN {X 0,Y 244.042,Z 354.827,A -85,B 0,C 180,E1 -19852.623,E2 -19852.623} C_VEL
LIN {X 0,Y 249.052,Z 365.513,A -85,B 0,C 180,E1 -19854.19,E2 -19854.19} C_VEL
LIN {X 0,Y 251.995,Z 372.73,A -85,B 0,C 180,E1 -19855.097,E2 -19855.097} C_VEL
LIN {X 0,Y 254.258,Z 390.589,A -85,B 0,C 180,E1 -19856.252,E2 -19856.252} C_VEL
LIN {X 0,Y 251.429,Z 443.241,A -85,B 0,C 180,E1 -19857.883,E2 -19857.883} C_VEL
LIN {X 0,Y 249.927,Z 456.228,A -85,B 0,C 180,E1 -19858.543,E2 -19858.543} C_VEL
LIN {X 0,Y 247.921,Z 468.437,A -85,B 0,C 180,E1 -19859.445,E2 -19859.445} C_VEL
LIN {X 0,Y 245.429,Z 480.282,A -85,B 0,C 180,E1 -19860.643,E2 -19860.643} C_VEL
LIN {X 0,Y 242.73,Z 491.657,A -85,B 0,C 180,E1 -19862.176,E2 -19862.176} C_VEL
LIN {X 0,Y 239.531,Z 503.046,A -85,B 0,C 180,E1 -19864.131,E2 -19864.131} C_VEL
LIN {X 0,Y 236.454,Z 513.02,A -85,B 0,C 180,E1 -19866.351,E2 -19866.351} C_VEL
LIN {X 0,Y 233.509,Z 522.068,A -85,B 0,C 180,E1 -19868.911,E2 -19868.911} C_VEL
LIN {X 0,Y 230.834,Z 529.97,A -85,B 0,C 180,E1 -19871.823,E2 -19871.823} C_VEL
LIN {X 0,Y 228.539,Z 536.305,A -85,B 0,C 180,E1 -19874.854,E2 -19874.854} C_VEL
LIN {X 0,Y 227.203,Z 540.462,A -85,B 0,C 180,E1 -19877.502,E2 -19877.502} C_VEL
LIN {X 0,Y 226.568,Z 542.656,A -85,B 0,C 180,E1 -19879.28,E2 -19879.28} C_VEL
LIN {X 0,Y 226.126,Z 544.402,A -85,B 0,C 180,E1 -19881.066,E2 -19881.066} C_VEL
LIN {X 0,Y 225.644,Z 546.703,A -85,B 0,C 180,E1 -19884.645,E2 -19884.645} C_VEL
LIN {X 0,Y 225.612,Z 547.231,A -85,B 0,C 180,E1 -19886.434,E2 -19886.434} C_VEL
LIN {X 0,Y 225.719,Z 547.348,A -85,B 0,C 180,E1 -19888.222,E2 -19888.222} C_VEL
LIN {X 0,Y 225.819,Z 547.072,A -85,B 0,C 180,E1 -19890.006,E2 -19890.006} C_VEL
LIN {X 0,Y 225.735,Z 546.39,A -85,B 0,C 180,E1 -19891.79,E2 -19891.79} C_VEL
LIN {X 0,Y 225.684,Z 544.273,A -85,B 0,C 180,E1 -19894.787,E2 -19894.787} C_VEL
LIN {X 0,Y 225.949,Z 540.514,A -85,B 0,C 180,E1 -19898.051,E2 -19898.051} C_VEL
LIN {X 0,Y 226.477,Z 536.227,A -85,B 0,C 180,E1 -19900.736,E2 -19900.736} C_VEL
LIN {X 0,Y 227.548,Z 529.692,A -85,B 0,C 180,E1 -19903.854,E2 -19903.854} C_VEL
LIN {X 0,Y 228.991,Z 522.503,A -85,B 0,C 180,E1 -19906.498,E2 -19906.498} C_VEL
LIN {X 0,Y 230.455,Z 515.7,A -85,B 0,C 180,E1 -19908.533,E2 -19908.533} C_VEL
LIN {X 0,Y 232.283,Z 506.26,A -85,B 0,C 180,E1 -19910.829,E2 -19910.829} C_VEL
LIN {X 0,Y 234.244,Z 496.499,A -85,B 0,C 180,E1 -19912.728,E2 -19912.728} C_VEL
LIN {X 0,Y 236.175,Z 485.828,A -85,B 0,C 180,E1 -19914.391,E2 -19914.391} C_VEL
LIN {X 0,Y 238.022,Z 473.93,A -85,B 0,C 180,E1 -19915.822,E2 -19915.822} C_VEL
LIN {X 0,Y 239.655,Z 461.659,A -85,B 0,C 180,E1 -19916.922,E2 -19916.922} C_VEL
LIN {X 0,Y 240.987,Z 448.267,A -85,B 0,C 180,E1 -19917.76,E2 -19917.76} C_VEL
LIN {X 0,Y 241.82,Z 431.812,A -85,B 0,C 180,E1 -19918.365,E2 -19918.365} C_VEL
LIN {X 0,Y 243.429,Z 387.974,A -85,B 0,C 180,E1 -19919.717,E2 -19919.717} C_VEL
LIN {X 0,Y 239.551,Z 358.297,A -85,B 0,C 180,E1 -19921.197,E2 -19921.197} C_VEL
LIN {X 0,Y 236.064,Z 348.343,A -85,B 0,C 180,E1 -19921.973,E2 -19921.973} C_VEL
LIN {X 0,Y 230.804,Z 334.958,A -85,B 0,C 180,E1 -19923.178,E2 -19923.178} C_VEL
LIN {X 0,Y 228.463,Z 324.443,A -85,B 0,C 180,E1 -19927.651,E2 -19927.651} C_VEL
LIN {X 0,Y 227.893,Z 322.095,A -85,B 0,C 180,E1 -19928.751,E2 -19928.751} C_VEL
LIN {X 0,Y 227.814,Z 322.106,A -85,B 0,C 180,E1 -19932.746,E2 -19932.746} C_VEL
LIN {X 0,Y 227.811,Z 322.109,A -85,B 0,C 180,E1 -19937.258,E2 -19937.258} C_VEL
LIN {X 0,Y 227.848,Z 322.103,A -85,B 0,C 180,E1 -19941.91,E2 -19941.91} C_VEL
LIN {X 0,Y 227.886,Z 322.099,A -85,B 0,C 180,E1 -19946.379,E2 -19946.379} C_VEL
LIN {X 0,Y 227.91,Z 322.093,A -85,B 0,C 180,E1 -19950.436,E2 -19950.436} C_VEL
LIN {X 0,Y 227.931,Z 322.09,A -85,B 0,C 180,E1 -19954.426,E2 -19954.426} C_VEL
LIN {X 0,Y 227.925,Z 322.092,A -85,B 0,C 180,E1 -19958.283,E2 -19958.283} C_VEL
LIN {X 0,Y 228.023,Z 322.057,A -85,B 0,C 180,E1 -19963.895,E2 -19963.895} C_VEL
LIN {X 0,Y 228.058,Z 322.074,A -85,B 0,C 180,E1 -19967.542,E2 -19967.542} C_VEL
LIN {X 0,Y 228.259,Z 322.053,A -85,B 0,C 180,E1 -19971.144,E2 -19971.144} C_VEL
LIN {X 0,Y 228.324,Z 322.04,A -85,B 0,C 180,E1 -19972.928,E2 -19972.928} C_VEL
LIN {X 0,Y 228.554,Z 321.983,A -85,B 0,C 180,E1 -19978.238,E2 -19978.238} C_VEL
LIN {X 0,Y 228.552,Z 322.005,A -85,B 0,C 180,E1 -19981.762,E2 -19981.762} C_VEL
LIN {X 0,Y 228.297,Z 322.046,A -85,B 0,C 180,E1 -19987.073,E2 -19987.073} C_VEL
LIN {X 0,Y 228.133,Z 322.058,A -85,B 0,C 180,E1 -19990.652,E2 -19990.652} C_VEL
LIN {X 0,Y 228.023,Z 322.079,A -85,B 0,C 180,E1 -19996.105,E2 -19996.105} C_VEL
LIN {X 0,Y 227.925,Z 322.09,A -85,B 0,C 180,E1 -20001.717,E2 -20001.717} C_VEL
LIN {X 0,Y 227.876,Z 322.09,A -85,B 0,C 180,E1 -20006.564,E2 -20006.564} C_VEL
LIN {X 0,Y 227.861,Z 322.069,A -85,B 0,C 180,E1 -20010.271,E2 -20010.271} C_VEL
LIN {X 0,Y 227.875,Z 322.079,A -85,B 0,C 180,E1 -20013.721,E2 -20013.721} C_VEL
LIN {X 0,Y 227.845,Z 322.102,A -85,B 0,C 180,E1 -20018.091,E2 -20018.091} C_VEL
LIN {X 0,Y 227.782,Z 322.106,A -85,B 0,C 180,E1 -20022.749,E2 -20022.749} C_VEL
LIN {X 0,Y 227.811,Z 322.106,A -85,B 0,C 180,E1 -20025.199,E2 -20025.199} C_VEL
LIN {X 0,Y 227.802,Z 322.102,A -85,B 0,C 180,E1 -20029.614,E2 -20029.614} C_VEL
LIN {X 0,Y 227.866,Z 322.1,A -85,B 0,C 180,E1 -20034.121,E2 -20034.121} C_VEL
LIN {X 0,Y 227.847,Z 322.105,A -85,B 0,C 180,E1 -20038.37,E2 -20038.37} C_VEL
LIN {X 0,Y 227.859,Z 322.102,A -85,B 0,C 180,E1 -20042.437,E2 -20042.437} C_VEL
LIN {X 0,Y 227.897,Z 322.095,A -85,B 0,C 180,E1 -20046.361,E2 -20046.361} C_VEL
LIN {X 0,Y 227.904,Z 322.096,A -85,B 0,C 180,E1 -20050.166,E2 -20050.166} C_VEL
LIN {X 0,Y 228.027,Z 322.08,A -85,B 0,C 180,E1 -20053.891,E2 -20053.891} C_VEL
LIN {X 0,Y 228.062,Z 322.075,A -85,B 0,C 180,E1 -20057.538,E2 -20057.538} C_VEL
LIN {X 0,Y 228.258,Z 322.049,A -85,B 0,C 180,E1 -20061.139,E2 -20061.139} C_VEL
LIN {X 0,Y 228.304,Z 322.045,A -85,B 0,C 180,E1 -20062.922,E2 -20062.922} C_VEL
LIN {X 0,Y 228.525,Z 322.016,A -85,B 0,C 180,E1 -20068.727,E2 -20068.727} C_VEL
LIN {X 0,Y 229.627,Z 325.029,A -85,B 0,C 180,E1 -20069.009,E2 -20069.009} C_VEL
LIN {X 0,Y 234.933,Z 336.029,A -85,B 0,C 180,E1 -20070.091,E2 -20070.091} C_VEL
LIN {X 0,Y 242.579,Z 355.878,A -85,B 0,C 180,E1 -20071.709,E2 -20071.709} C_VEL
LIN {X 0,Y 244.316,Z 360.831,A -85,B 0,C 180,E1 -20072.077,E2 -20072.077} C_VEL
LIN {X 0,Y 241.582,Z 427.472,A -85,B 0,C 180,E1 -20074.155,E2 -20074.155} C_VEL
LIN {X 0,Y 240.552,Z 441.207,A -85,B 0,C 180,E1 -20074.928,E2 -20074.928} C_VEL
LIN {X 0,Y 239.26,Z 453.752,A -85,B 0,C 180,E1 -20075.976,E2 -20075.976} C_VEL
LIN {X 0,Y 237.508,Z 466.502,A -85,B 0,C 180,E1 -20077.432,E2 -20077.432} C_VEL
LIN {X 0,Y 235.515,Z 478.063,A -85,B 0,C 180,E1 -20079.142,E2 -20079.142} C_VEL
LIN {X 0,Y 233.383,Z 489.226,A -85,B 0,C 180,E1 -20081.281,E2 -20081.281} C_VEL
LIN {X 0,Y 231.689,Z 497.909,A -85,B 0,C 180,E1 -20083.365,E2 -20083.365} C_VEL
LIN {X 0,Y 229.842,Z 506.628,A -85,B 0,C 180,E1 -20085.967,E2 -20085.967} C_VEL
LIN {X 0,Y 228.259,Z 514.18,A -85,B 0,C 180,E1 -20088.855,E2 -20088.855} C_VEL
LIN {X 0,Y 227.102,Z 520.176,A -85,B 0,C 180,E1 -20091.814,E2 -20091.814} C_VEL
LIN {X 0,Y 226.333,Z 524.563,A -85,B 0,C 180,E1 -20094.706,E2 -20094.706} C_VEL
LIN {X 0,Y 225.621,Z 527.92,A -85,B 0,C 180,E1 -20097.847,E2 -20097.847} C_VEL
LIN {X 0,Y 225.402,Z 529.427,A -85,B 0,C 180,E1 -20099.917,E2 -20099.917} C_VEL
LIN {X 0,Y 225.385,Z 530.542,A -85,B 0,C 180,E1 -20102.656,E2 -20102.656} C_VEL
LIN {X 0,Y 225.685,Z 530.658,A -85,B 0,C 180,E1 -20105.937,E2 -20105.937} C_VEL
LIN {X 0,Y 226.357,Z 529.48,A -85,B 0,C 180,E1 -20109.085,E2 -20109.085} C_VEL
LIN {X 0,Y 227.445,Z 527.13,A -85,B 0,C 180,E1 -20112.132,E2 -20112.132} C_VEL
LIN {X 0,Y 228.82,Z 523.674,A -85,B 0,C 180,E1 -20115.055,E2 -20115.055} C_VEL
LIN {X 0,Y 230.637,Z 519.011,A -85,B 0,C 180,E1 -20117.903,E2 -20117.903} C_VEL
LIN {X 0,Y 232.937,Z 512.98,A -85,B 0,C 180,E1 -20120.684,E2 -20120.684} C_VEL
LIN {X 0,Y 235.713,Z 505.306,A -85,B 0,C 180,E1 -20123.393,E2 -20123.393} C_VEL
LIN {X 0,Y 238.365,Z 497.317,A -85,B 0,C 180,E1 -20125.63,E2 -20125.63} C_VEL
LIN {X 0,Y 241.105,Z 488.18,A -85,B 0,C 180,E1 -20127.69,E2 -20127.69} C_VEL
LIN {X 0,Y 243.939,Z 477.995,A -85,B 0,C 180,E1 -20129.49,E2 -20129.49} C_VEL
LIN {X 0,Y 246.44,Z 467.272,A -85,B 0,C 180,E1 -20131,E2 -20131} C_VEL
LIN {X 0,Y 248.869,Z 454.738,A -85,B 0,C 180,E1 -20132.359,E2 -20132.359} C_VEL
LIN {X 0,Y 250.722,Z 441.614,A -85,B 0,C 180,E1 -20133.391,E2 -20133.391} C_VEL
LIN {X 0,Y 251.991,Z 429.334,A -85,B 0,C 180,E1 -20134.044,E2 -20134.044} C_VEL
LIN {X 0,Y 255.235,Z 371.174,A -85,B 0,C 180,E1 -20135.826,E2 -20135.826} C_VEL
LIN {X 0,Y 255.211,Z 369.521,A -85,B 0,C 180,E1 -20135.897,E2 -20135.897} C_VEL
LIN {X 0,Y 250.287,Z 358.451,A -85,B 0,C 180,E1 -20137.34,E2 -20137.34} C_VEL
LIN {X 0,Y 244.809,Z 347.925,A -85,B 0,C 180,E1 -20138.998,E2 -20138.998} C_VEL
LIN {X 0,Y 239.813,Z 339.735,A -85,B 0,C 180,E1 -20140.583,E2 -20140.583} C_VEL
LIN {X 0,Y 236.658,Z 335.183,A -85,B 0,C 180,E1 -20141.628,E2 -20141.628} C_VEL
LIN {X 0,Y 234.073,Z 331.475,A -85,B 0,C 180,E1 -20142.527,E2 -20142.527} C_VEL
LIN {X 0,Y 231.808,Z 328.291,A -85,B 0,C 180,E1 -20143.342,E2 -20143.342} C_VEL
LIN {X 0,Y 231.134,Z 327.126,A -85,B 0,C 180,E1 -20143.602,E2 -20143.602} C_VEL
LIN {X 0,Y 229.001,Z 324.914,A -85,B 0,C 180,E1 -20144.366,E2 -20144.366} C_VEL
LIN {X 0,Y 228,Z 322.086,A -85,B 0,C 180,E1 -20144.868,E2 -20144.868} C_VEL
LIN {X 0,Y 228.177,Z 322.058,A -85,B 0,C 180,E1 -20150.215,E2 -20150.215} C_VEL
LIN {X 0,Y 228.28,Z 322.042,A -85,B 0,C 180,E1 -20152.926,E2 -20152.926} C_VEL
LIN {X 0,Y 228.512,Z 322.019,A -85,B 0,C 180,E1 -20158.238,E2 -20158.238} C_VEL
LIN {X 0,Y 228.513,Z 322.02,A -85,B 0,C 180,E1 -20161.762,E2 -20161.762} C_VEL
LIN {X 0,Y 228.29,Z 322.038,A -85,B 0,C 180,E1 -20167.073,E2 -20167.073} C_VEL
LIN {X 0,Y 228.074,Z 322.066,A -85,B 0,C 180,E1 -20171.145,E2 -20171.145} C_VEL
LIN {X 0,Y 228.008,Z 322.069,A -85,B 0,C 180,E1 -20176.106,E2 -20176.106} C_VEL
LIN {X 0,Y 227.923,Z 322.081,A -85,B 0,C 180,E1 -20178.821,E2 -20178.821} C_VEL
LIN {X 0,Y 227.239,Z 322.166,A -85,B 0,C 180,E1 -20180.295,E2 -20180.295} C_VEL
LIN {X 0,Y 224.396,Z 322.53,A -85,B 0,C 180,E1 -20182.701,E2 -20182.701} C_VEL
LIN {X 0,Y 221.986,Z 322.835,A -85,B 0,C 180,E1 -20184.665,E2 -20184.665} C_VEL
LIN {X 0,Y 220.945,Z 322.961,A -85,B 0,C 180,E1 -20186.188,E2 -20186.188} C_VEL
LIN {X 0,Y 220.856,Z 322.969,A -85,B 0,C 180,E1 -20186.705,E2 -20186.705} C_VEL
LIN {X 0,Y 220.808,Z 322.975,A -85,B 0,C 180,E1 -20190.772,E2 -20190.772} C_VEL
LIN {X 0,Y 220.788,Z 322.976,A -85,B 0,C 180,E1 -20194.957,E2 -20194.957} C_VEL
LIN {X 0,Y 220.855,Z 322.976,A -85,B 0,C 180,E1 -20199.527,E2 -20199.527} C_VEL
LIN {X 0,Y 220.861,Z 323.049,A -85,B 0,C 180,E1 -20200.068,E2 -20200.068} C_VEL
LIN {X 0,Y 222.694,Z 328.637,A -85,B 0,C 180,E1 -20203.972,E2 -20203.972} C_VEL
LIN {X 0,Y 223.633,Z 331.498,A -85,B 0,C 180,E1 -20205.733,E2 -20205.733} C_VEL
LIN {X 0,Y 226.873,Z 336.574,A -85,B 0,C 180,E1 -20207.099,E2 -20207.099} C_VEL
LIN {X 0,Y 231.765,Z 344.56,A -85,B 0,C 180,E1 -20208.982,E2 -20208.982} C_VEL
LIN {X 0,Y 235.203,Z 350.526,A -85,B 0,C 180,E1 -20210.235,E2 -20210.235} C_VEL
LIN {X 0,Y 240.867,Z 361.571,A -85,B 0,C 180,E1 -20212.19,E2 -20212.19} C_VEL
LIN {X 0,Y 246.59,Z 374.691,A -85,B 0,C 180,E1 -20214.059,E2 -20214.059} C_VEL
LIN {X 0,Y 247.888,Z 382.943,A -85,B 0,C 180,E1 -20214.687,E2 -20214.687} C_VEL
LIN {X 0,Y 248.796,Z 391.741,A -85,B 0,C 180,E1 -20215.247,E2 -20215.247} C_VEL
LIN {X 0,Y 245.923,Z 442.507,A -85,B 0,C 180,E1 -20216.835,E2 -20216.835} C_VEL
LIN {X 0,Y 244.279,Z 456.303,A -85,B 0,C 180,E1 -20217.546,E2 -20217.546} C_VEL
LIN {X 0,Y 242.091,Z 468.939,A -85,B 0,C 180,E1 -20218.505,E2 -20218.505} C_VEL
LIN {X 0,Y 239.317,Z 481.361,A -85,B 0,C 180,E1 -20219.816,E2 -20219.816} C_VEL
LIN {X 0,Y 236.526,Z 492.495,A -85,B 0,C 180,E1 -20221.38,E2 -20221.38} C_VEL
LIN {X 0,Y 233.534,Z 502.623,A -85,B 0,C 180,E1 -20223.174,E2 -20223.174} C_VEL
LIN {X 0,Y 230.531,Z 511.784,A -85,B 0,C 180,E1 -20225.225,E2 -20225.225} C_VEL
LIN {X 0,Y 227.409,Z 520.746,A -85,B 0,C 180,E1 -20227.762,E2 -20227.762} C_VEL
LIN {X 0,Y 224.785,Z 528.021,A -85,B 0,C 180,E1 -20230.368,E2 -20230.368} C_VEL
LIN {X 0,Y 222.985,Z 532.965,A -85,B 0,C 180,E1 -20232.585,E2 -20232.585} C_VEL
LIN {X 0,Y 221.086,Z 537.802,A -85,B 0,C 180,E1 -20235.275,E2 -20235.275} C_VEL
LIN {X 0,Y 219.872,Z 541.537,A -85,B 0,C 180,E1 -20238.015,E2 -20238.015} C_VEL
LIN {X 0,Y 219.078,Z 544.273,A -85,B 0,C 180,E1 -20240.777,E2 -20240.777} C_VEL
LIN {X 0,Y 218.566,Z 546.499,A -85,B 0,C 180,E1 -20244.471,E2 -20244.471} C_VEL
LIN {X 0,Y 218.63,Z 547.067,A -85,B 0,C 180,E1 -20248.164,E2 -20248.164} C_VEL
LIN {X 0,Y 218.751,Z 546.764,A -85,B 0,C 180,E1 -20250.006,E2 -20250.006} C_VEL
LIN {X 0,Y 218.647,Z 546.047,A -85,B 0,C 180,E1 -20251.848,E2 -20251.848} C_VEL
LIN {X 0,Y 218.584,Z 544.125,A -85,B 0,C 180,E1 -20254.637,E2 -20254.637} C_VEL
LIN {X 0,Y 218.778,Z 541.24,A -85,B 0,C 180,E1 -20257.388,E2 -20257.388} C_VEL
LIN {X 0,Y 219.246,Z 537.266,A -85,B 0,C 180,E1 -20260.16,E2 -20260.16} C_VEL
LIN {X 0,Y 220.219,Z 531.104,A -85,B 0,C 180,E1 -20263.383,E2 -20263.383} C_VEL
LIN {X 0,Y 221.654,Z 524.348,A -85,B 0,C 180,E1 -20266.112,E2 -20266.112} C_VEL
LIN {X 0,Y 223.368,Z 516.388,A -85,B 0,C 180,E1 -20268.678,E2 -20268.678} C_VEL
LIN {X 0,Y 225.216,Z 507.249,A -85,B 0,C 180,E1 -20271.035,E2 -20271.035} C_VEL
LIN {X 0,Y 227.135,Z 497.724,A -85,B 0,C 180,E1 -20272.999,E2 -20272.999} C_VEL
LIN {X 0,Y 229.158,Z 487.377,A -85,B 0,C 180,E1 -20274.704,E2 -20274.704} C_VEL
LIN {X 0,Y 231.076,Z 476.075,A -85,B 0,C 180,E1 -20276.172,E2 -20276.172} C_VEL
LIN {X 0,Y 232.841,Z 463.354,A -85,B 0,C 180,E1 -20277.411,E2 -20277.411} C_VEL
LIN {X 0,Y 234.297,Z 449.928,A -85,B 0,C 180,E1 -20278.319,E2 -20278.319} C_VEL
LIN {X 0,Y 235.112,Z 437.108,A -85,B 0,C 180,E1 -20278.867,E2 -20278.867} C_VEL
LIN {X 0,Y 236.919,Z 388.544,A -85,B 0,C 180,E1 -20280.411,E2 -20280.411} C_VEL
LIN {X 0,Y 233.279,Z 360.126,A -85,B 0,C 180,E1 -20281.874,E2 -20281.874} C_VEL
LIN {X 0,Y 227.418,Z 344.457,A -85,B 0,C 180,E1 -20283.194,E2 -20283.194} C_VEL
LIN {X 0,Y 223.531,Z 334.773,A -85,B 0,C 180,E1 -20284.114,E2 -20284.114} C_VEL
LIN {X 0,Y 221.503,Z 325.701,A -85,B 0,C 180,E1 -20288.123,E2 -20288.123} C_VEL
LIN {X 0,Y 220.855,Z 322.971,A -85,B 0,C 180,E1 -20289.389,E2 -20289.389} C_VEL
LIN {X 0,Y 220.775,Z 322.989,A -85,B 0,C 180,E1 -20294.458,E2 -20294.458} C_VEL
LIN {X 0,Y 220.77,Z 322.987,A -85,B 0,C 180,E1 -20298.047,E2 -20298.047} C_VEL
LIN {X 0,Y 220.834,Z 322.979,A -85,B 0,C 180,E1 -20302.795,E2 -20302.795} C_VEL
LIN {X 0,Y 220.823,Z 322.98,A -85,B 0,C 180,E1 -20307.245,E2 -20307.245} C_VEL
LIN {X 0,Y 220.833,Z 322.977,A -85,B 0,C 180,E1 -20311.486,E2 -20311.486} C_VEL
LIN {X 0,Y 220.866,Z 322.97,A -85,B 0,C 180,E1 -20315.565,E2 -20315.565} C_VEL
LIN {X 0,Y 220.857,Z 322.969,A -85,B 0,C 180,E1 -20319.51,E2 -20319.51} C_VEL
LIN {X 0,Y 220.982,Z 322.932,A -85,B 0,C 180,E1 -20323.368,E2 -20323.368} C_VEL
LIN {X 0,Y 221.067,Z 322.946,A -85,B 0,C 180,E1 -20329.004,E2 -20329.004} C_VEL
LIN {X 0,Y 221.258,Z 322.92,A -85,B 0,C 180,E1 -20332.701,E2 -20332.701} C_VEL
LIN {X 0,Y 221.488,Z 322.86,A -85,B 0,C 180,E1 -20338.182,E2 -20338.182} C_VEL
LIN {X 0,Y 221.51,Z 322.881,A -85,B 0,C 180,E1 -20341.818,E2 -20341.818} C_VEL
LIN {X 0,Y 221.235,Z 322.927,A -85,B 0,C 180,E1 -20347.3,E2 -20347.3} C_VEL
LIN {X 0,Y 221.059,Z 322.939,A -85,B 0,C 180,E1 -20350.997,E2 -20350.997} C_VEL
LIN {X 0,Y 220.982,Z 322.954,A -85,B 0,C 180,E1 -20356.633,E2 -20356.633} C_VEL
LIN {X 0,Y 220.853,Z 322.97,A -85,B 0,C 180,E1 -20360.49,E2 -20360.49} C_VEL
LIN {X 0,Y 220.808,Z 322.977,A -85,B 0,C 180,E1 -20364.442,E2 -20364.442} C_VEL
LIN {X 0,Y 220.79,Z 322.962,A -85,B 0,C 180,E1 -20368.52,E2 -20368.52} C_VEL
LIN {X 0,Y 220.809,Z 322.95,A -85,B 0,C 180,E1 -20372.758,E2 -20372.758} C_VEL
LIN {X 0,Y 220.804,Z 322.977,A -85,B 0,C 180,E1 -20377.271,E2 -20377.271} C_VEL
LIN {X 0,Y 220.748,Z 322.984,A -85,B 0,C 180,E1 -20381.958,E2 -20381.958} C_VEL
LIN {X 0,Y 220.754,Z 322.985,A -85,B 0,C 180,E1 -20385.537,E2 -20385.537} C_VEL
LIN {X 0,Y 220.787,Z 322.978,A -85,B 0,C 180,E1 -20390.455,E2 -20390.455} C_VEL
LIN {X 0,Y 220.834,Z 322.98,A -85,B 0,C 180,E1 -20392.79,E2 -20392.79} C_VEL
LIN {X 0,Y 220.81,Z 322.982,A -85,B 0,C 180,E1 -20397.238,E2 -20397.238} C_VEL
LIN {X 0,Y 220.808,Z 322.98,A -85,B 0,C 180,E1 -20401.478,E2 -20401.478} C_VEL
LIN {X 0,Y 220.852,Z 322.974,A -85,B 0,C 180,E1 -20405.559,E2 -20405.559} C_VEL
LIN {X 0,Y 220.861,Z 322.975,A -85,B 0,C 180,E1 -20409.506,E2 -20409.506} C_VEL
LIN {X 0,Y 220.984,Z 322.96,A -85,B 0,C 180,E1 -20413.363,E2 -20413.363} C_VEL
LIN {X 0,Y 221.068,Z 322.947,A -85,B 0,C 180,E1 -20418.998,E2 -20418.998} C_VEL
LIN {X 0,Y 221.242,Z 322.924,A -85,B 0,C 180,E1 -20422.695,E2 -20422.695} C_VEL
LIN {X 0,Y 221.403,Z 322.904,A -85,B 0,C 180,E1 -20427.777,E2 -20427.777} C_VEL
LIN {X 0,Y 222.514,Z 325.802,A -85,B 0,C 180,E1 -20428.075,E2 -20428.075} C_VEL
LIN {X 0,Y 228.975,Z 338.878,A -85,B 0,C 180,E1 -20429.451,E2 -20429.451} C_VEL
LIN {X 0,Y 236.696,Z 359.132,A -85,B 0,C 180,E1 -20431.144,E2 -20431.144} C_VEL
LIN {X 0,Y 237.876,Z 363.05,A -85,B 0,C 180,E1 -20431.424,E2 -20431.424} C_VEL
LIN {X 0,Y 235.083,Z 427.483,A -85,B 0,C 180,E1 -20433.476,E2 -20433.476} C_VEL
LIN {X 0,Y 234.037,Z 440.983,A -85,B 0,C 180,E1 -20434.246,E2 -20434.246} C_VEL
LIN {X 0,Y 232.74,Z 453.472,A -85,B 0,C 180,E1 -20435.3,E2 -20435.3} C_VEL
LIN {X 0,Y 231.208,Z 464.443,A -85,B 0,C 180,E1 -20436.539,E2 -20436.539} C_VEL
LIN {X 0,Y 229.294,Z 475.542,A -85,B 0,C 180,E1 -20438.143,E2 -20438.143} C_VEL
LIN {X 0,Y 227.224,Z 486.232,A -85,B 0,C 180,E1 -20440.099,E2 -20440.099} C_VEL
LIN {X 0,Y 225.383,Z 495.184,A -85,B 0,C 180,E1 -20442.144,E2 -20442.144} C_VEL
LIN {X 0,Y 223.579,Z 503.677,A -85,B 0,C 180,E1 -20444.558,E2 -20444.558} C_VEL
LIN {X 0,Y 221.955,Z 511.184,A -85,B 0,C 180,E1 -20447.222,E2 -20447.222} C_VEL
LIN {X 0,Y 220.692,Z 517.415,A -85,B 0,C 180,E1 -20450.012,E2 -20450.012} C_VEL
LIN {X 0,Y 219.797,Z 521.891,A -85,B 0,C 180,E1 -20452.555,E2 -20452.555} C_VEL
LIN {X 0,Y 219.247,Z 524.811,A -85,B 0,C 180,E1 -20454.619,E2 -20454.619} C_VEL
LIN {X 0,Y 218.748,Z 527.145,A -85,B 0,C 180,E1 -20456.722,E2 -20456.722} C_VEL
LIN {X 0,Y 218.345,Z 529.461,A -85,B 0,C 180,E1 -20459.649,E2 -20459.649} C_VEL
LIN {X 0,Y 218.305,Z 530.893,A -85,B 0,C 180,E1 -20463.172,E2 -20463.172} C_VEL
LIN {X 0,Y 218.674,Z 530.862,A -85,B 0,C 180,E1 -20466.536,E2 -20466.536} C_VEL
LIN {X 0,Y 219.464,Z 529.566,A -85,B 0,C 180,E1 -20469.816,E2 -20469.816} C_VEL
LIN {X 0,Y 220.681,Z 527.146,A -85,B 0,C 180,E1 -20472.905,E2 -20472.905} C_VEL
LIN {X 0,Y 222.17,Z 523.61,A -85,B 0,C 180,E1 -20475.898,E2 -20475.898} C_VEL
LIN {X 0,Y 224.13,Z 518.854,A -85,B 0,C 180,E1 -20478.815,E2 -20478.815} C_VEL
LIN {X 0,Y 226.672,Z 512.625,A -85,B 0,C 180,E1 -20481.676,E2 -20481.676} C_VEL
LIN {X 0,Y 229.691,Z 504.801,A -85,B 0,C 180,E1 -20484.454,E2 -20484.454} C_VEL
LIN {X 0,Y 232.575,Z 496.612,A -85,B 0,C 180,E1 -20486.747,E2 -20486.747} C_VEL
LIN {X 0,Y 235.667,Z 486.418,A -85,B 0,C 180,E1 -20489.006,E2 -20489.006} C_VEL
LIN {X 0,Y 238.597,Z 476.181,A -85,B 0,C 180,E1 -20490.764,E2 -20490.764} C_VEL
LIN {X 0,Y 241.362,Z 464.275,A -85,B 0,C 180,E1 -20492.377,E2 -20492.377} C_VEL
LIN {X 0,Y 243.797,Z 451.428,A -85,B 0,C 180,E1 -20493.668,E2 -20493.668} C_VEL
LIN {X 0,Y 245.478,Z 438.714,A -85,B 0,C 180,E1 -20494.613,E2 -20494.613} C_VEL
LIN {X 0,Y 246.76,Z 426.123,A -85,B 0,C 180,E1 -20495.191,E2 -20495.191} C_VEL
LIN {X 0,Y 249.714,Z 371.705,A -85,B 0,C 180,E1 -20496.897,E2 -20496.897} C_VEL
LIN {X 0,Y 244.894,Z 360.815,A -85,B 0,C 180,E1 -20498.407,E2 -20498.407} C_VEL
LIN {X 0,Y 240.002,Z 351.59,A -85,B 0,C 180,E1 -20499.972,E2 -20499.972} C_VEL
LIN {X 0,Y 235.52,Z 344.231,A -85,B 0,C 180,E1 -20501.478,E2 -20501.478} C_VEL
LIN {X 0,Y 230.429,Z 336.812,A -85,B 0,C 180,E1 -20503.292,E2 -20503.292} C_VEL
LIN {X 0,Y 227.604,Z 332.741,A -85,B 0,C 180,E1 -20504.371,E2 -20504.371} C_VEL
LIN {X 0,Y 225.332,Z 329.794,A -85,B 0,C 180,E1 -20505.272,E2 -20505.272} C_VEL
LIN {X 0,Y 224.577,Z 328.294,A -85,B 0,C 180,E1 -20505.617,E2 -20505.617} C_VEL
LIN {X 0,Y 222.331,Z 326.37,A -85,B 0,C 180,E1 -20506.519,E2 -20506.519} C_VEL
LIN {X 0,Y 221.075,Z 323.665,A -85,B 0,C 180,E1 -20507.142,E2 -20507.142} C_VEL
LIN {X 0,Y 220.956,Z 322.958,A -85,B 0,C 180,E1 -20507.252,E2 -20507.252} C_VEL
LIN {X 0,Y 221.151,Z 322.938,A -85,B 0,C 180,E1 -20510.857,E2 -20510.857} C_VEL
LIN {X 0,Y 221.214,Z 322.921,A -85,B 0,C 180,E1 -20512.699,E2 -20512.699} C_VEL
LIN {X 0,Y 221.47,Z 322.897,A -85,B 0,C 180,E1 -20518.181,E2 -20518.181} C_VEL
LIN {X 0,Y 221.471,Z 322.897,A -85,B 0,C 180,E1 -20521.818,E2 -20521.818} C_VEL
LIN {X 0,Y 221.226,Z 322.917,A -85,B 0,C 180,E1 -20527.3,E2 -20527.3} C_VEL
LIN {X 0,Y 221.051,Z 322.942,A -85,B 0,C 180,E1 -20530.997,E2 -20530.997} C_VEL
LIN {X 0,Y 220.973,Z 322.945,A -85,B 0,C 180,E1 -20536.633,E2 -20536.633} C_VEL
LIN {X 0,Y 220.887,Z 322.954,A -85,B 0,C 180,E1 -20540.487,E2 -20540.487} C_VEL
LIN {X 0,Y 220.846,Z 322.96,A -85,B 0,C 180,E1 -20544.438,E2 -20544.438} C_VEL
LIN {X 0,Y 220.856,Z 322.969,A -85,B 0,C 180,E1 -20546.705,E2 -20546.705} C_VEL
LIN {X 0,Y 220.183,Z 323.048,A -85,B 0,C 180,E1 -20548.226,E2 -20548.226} C_VEL
LIN {X 0,Y 217.358,Z 323.406,A -85,B 0,C 180,E1 -20550.711,E2 -20550.711} C_VEL
LIN {X 0,Y 214.106,Z 323.816,A -85,B 0,C 180,E1 -20553.782,E2 -20553.782} C_VEL
LIN {X 0,Y 213.749,Z 323.853,A -85,B 0,C 180,E1 -20554.847,E2 -20554.847} C_VEL
LIN {X 0,Y 213.784,Z 323.876,A -85,B 0,C 180,E1 -20557.545,E2 -20557.545} C_VEL
LIN {X 0,Y 215.668,Z 329.391,A -85,B 0,C 180,E1 -20561.915,E2 -20561.915} C_VEL
LIN {X 0,Y 216.236,Z 330.989,A -85,B 0,C 180,E1 -20562.962,E2 -20562.962} C_VEL
LIN {X 0,Y 219.394,Z 335.916,A -85,B 0,C 180,E1 -20564.491,E2 -20564.491} C_VEL
LIN {X 0,Y 220.955,Z 338.142,A -85,B 0,C 180,E1 -20565.197,E2 -20565.197} C_VEL
LIN {X 0,Y 224.862,Z 344.295,A -85,B 0,C 180,E1 -20566.891,E2 -20566.891} C_VEL
LIN {X 0,Y 230.599,Z 354.055,A -85,B 0,C 180,E1 -20569.149,E2 -20569.149} C_VEL
LIN {X 0,Y 236.185,Z 365.148,A -85,B 0,C 180,E1 -20571.205,E2 -20571.205} C_VEL
LIN {X 0,Y 241.796,Z 378.29,A -85,B 0,C 180,E1 -20573.161,E2 -20573.161} C_VEL
LIN {X 0,Y 243.295,Z 391.316,A -85,B 0,C 180,E1 -20574.07,E2 -20574.07} C_VEL
LIN {X 0,Y 243.284,Z 396.939,A -85,B 0,C 180,E1 -20574.314,E2 -20574.314} C_VEL
LIN {X 0,Y 240.425,Z 442.946,A -85,B 0,C 180,E1 -20575.782,E2 -20575.782} C_VEL
LIN {X 0,Y 238.719,Z 456.487,A -85,B 0,C 180,E1 -20576.504,E2 -20576.504} C_VEL
LIN {X 0,Y 236.577,Z 468.426,A -85,B 0,C 180,E1 -20577.432,E2 -20577.432} C_VEL
LIN {X 0,Y 233.679,Z 480.876,A -85,B 0,C 180,E1 -20578.757,E2 -20578.757} C_VEL
LIN {X 0,Y 230.717,Z 492.054,A -85,B 0,C 180,E1 -20580.339,E2 -20580.339} C_VEL
LIN {X 0,Y 227.591,Z 502.218,A -85,B 0,C 180,E1 -20582.165,E2 -20582.165} C_VEL
LIN {X 0,Y 224.13,Z 512.22,A -85,B 0,C 180,E1 -20584.467,E2 -20584.467} C_VEL
LIN {X 0,Y 220.859,Z 521.068,A -85,B 0,C 180,E1 -20587.065,E2 -20587.065} C_VEL
LIN {X 0,Y 218.116,Z 528.207,A -85,B 0,C 180,E1 -20589.742,E2 -20589.742} C_VEL
LIN {X 0,Y 215.494,Z 534.763,A -85,B 0,C 180,E1 -20592.939,E2 -20592.939} C_VEL
LIN {X 0,Y 213.704,Z 539.138,A -85,B 0,C 180,E1 -20595.728,E2 -20595.728} C_VEL
LIN {X 0,Y 212.568,Z 542.469,A -85,B 0,C 180,E1 -20598.565,E2 -20598.565} C_VEL
LIN {X 0,Y 212.051,Z 544.149,A -85,B 0,C 180,E1 -20600.468,E2 -20600.468} C_VEL
LIN {X 0,Y 211.665,Z 545.43,A -85,B 0,C 180,E1 -20602.375,E2 -20602.375} C_VEL
LIN {X 0,Y 211.418,Z 546.675,A -85,B 0,C 180,E1 -20605.765,E2 -20605.765} C_VEL
LIN {X 0,Y 211.542,Z 546.783,A -85,B 0,C 180,E1 -20608.102,E2 -20608.102} C_VEL
LIN {X 0,Y 211.662,Z 546.45,A -85,B 0,C 180,E1 -20610.006,E2 -20610.006} C_VEL
LIN {X 0,Y 211.561,Z 545.677,A -85,B 0,C 180,E1 -20611.91,E2 -20611.91} C_VEL
LIN {X 0,Y 211.509,Z 543.9,A -85,B 0,C 180,E1 -20614.555,E2 -20614.555} C_VEL
LIN {X 0,Y 211.702,Z 540.762,A -85,B 0,C 180,E1 -20617.637,E2 -20617.637} C_VEL
LIN {X 0,Y 212.205,Z 536.715,A -85,B 0,C 180,E1 -20620.501,E2 -20620.501} C_VEL
LIN {X 0,Y 213.29,Z 530.447,A -85,B 0,C 180,E1 -20623.826,E2 -20623.826} C_VEL
LIN {X 0,Y 214.776,Z 523.599,A -85,B 0,C 180,E1 -20626.643,E2 -20626.643} C_VEL
LIN {X 0,Y 216.59,Z 515.315,A -85,B 0,C 180,E1 -20629.35,E2 -20629.35} C_VEL
LIN {X 0,Y 218.542,Z 506.214,A -85,B 0,C 180,E1 -20631.71,E2 -20631.71} C_VEL
LIN {X 0,Y 220.633,Z 496.548,A -85,B 0,C 180,E1 -20633.718,E2 -20633.718} C_VEL
LIN {X 0,Y 222.662,Z 485.99,A -85,B 0,C 180,E1 -20635.476,E2 -20635.476} C_VEL
LIN {X 0,Y 224.39,Z 476.2,A -85,B 0,C 180,E1 -20636.763,E2 -20636.763} C_VEL
LIN {X 0,Y 226.206,Z 463.656,A -85,B 0,C 180,E1 -20638.033,E2 -20638.033} C_VEL
LIN {X 0,Y 227.701,Z 450.457,A -85,B 0,C 180,E1 -20638.964,E2 -20638.964} C_VEL
LIN {X 0,Y 228.629,Z 436.763,A -85,B 0,C 180,E1 -20639.574,E2 -20639.574} C_VEL
LIN {X 0,Y 230.512,Z 389.617,A -85,B 0,C 180,E1 -20641.107,E2 -20641.107} C_VEL
LIN {X 0,Y 226.973,Z 361.795,A -85,B 0,C 180,E1 -20642.583,E2 -20642.583} C_VEL
LIN {X 0,Y 218.962,Z 341.251,A -85,B 0,C 180,E1 -20644.462,E2 -20644.462} C_VEL
LIN {X 0,Y 216.227,Z 334.493,A -85,B 0,C 180,E1 -20645.152,E2 -20645.152} C_VEL
LIN {X 0,Y 214.394,Z 326.457,A -85,B 0,C 180,E1 -20648.846,E2 -20648.846} C_VEL
LIN {X 0,Y 213.77,Z 323.857,A -85,B 0,C 180,E1 -20650.151,E2 -20650.151} C_VEL
LIN {X 0,Y 213.712,Z 323.865,A -85,B 0,C 180,E1 -20653.682,E2 -20653.682} C_VEL
LIN {X 0,Y 213.712,Z 323.867,A -85,B 0,C 180,E1 -20656.347,E2 -20656.347} C_VEL
LIN {X 0,Y 213.717,Z 323.863,A -85,B 0,C 180,E1 -20659.148,E2 -20659.148} C_VEL
LIN {X 0,Y 213.75,Z 323.86,A -85,B 0,C 180,E1 -20663.713,E2 -20663.713} C_VEL
LIN {X 0,Y 213.789,Z 323.854,A -85,B 0,C 180,E1 -20668.733,E2 -20668.733} C_VEL
LIN {X 0,Y 213.836,Z 323.851,A -85,B 0,C 180,E1 -20672.604,E2 -20672.604} C_VEL
LIN {X 0,Y 213.808,Z 323.853,A -85,B 0,C 180,E1 -20676.987,E2 -20676.987} C_VEL
LIN {X 0,Y 213.891,Z 323.817,A -85,B 0,C 180,E1 -20682.799,E2 -20682.799} C_VEL
LIN {X 0,Y 213.937,Z 323.824,A -85,B 0,C 180,E1 -20686.706,E2 -20686.706} C_VEL
LIN {X 0,Y 214.135,Z 323.81,A -85,B 0,C 180,E1 -20690.555,E2 -20690.555} C_VEL
LIN {X 0,Y 214.097,Z 323.803,A -85,B 0,C 180,E1 -20694.348,E2 -20694.348} C_VEL
LIN {X 0,Y 214.425,Z 323.738,A -85,B 0,C 180,E1 -20698.122,E2 -20698.122} C_VEL
LIN {X 0,Y 214.542,Z 323.735,A -85,B 0,C 180,E1 -20700,E2 -20700} C_VEL
LIN {X 0,Y 214.443,Z 323.761,A -85,B 0,C 180,E1 -20701.878,E2 -20701.878} C_VEL
LIN {X 0,Y 214.177,Z 323.806,A -85,B 0,C 180,E1 -20707.542,E2 -20707.542} C_VEL
LIN {X 0,Y 213.992,Z 323.82,A -85,B 0,C 180,E1 -20711.365,E2 -20711.365} C_VEL
LIN {X 0,Y 213.889,Z 323.841,A -85,B 0,C 180,E1 -20715.24,E2 -20715.24} C_VEL
LIN {X 0,Y 213.798,Z 323.84,A -85,B 0,C 180,E1 -20719.191,E2 -20719.191} C_VEL
LIN {X 0,Y 213.792,Z 323.851,A -85,B 0,C 180,E1 -20723.233,E2 -20723.233} C_VEL
LIN {X 0,Y 213.775,Z 323.845,A -85,B 0,C 180,E1 -20727.416,E2 -20727.416} C_VEL
LIN {X 0,Y 213.726,Z 323.822,A -85,B 0,C 180,E1 -20731.745,E2 -20731.745} C_VEL
LIN {X 0,Y 213.748,Z 323.852,A -85,B 0,C 180,E1 -20736.288,E2 -20736.288} C_VEL
LIN {X 0,Y 213.702,Z 323.861,A -85,B 0,C 180,E1 -20741.128,E2 -20741.128} C_VEL
LIN {X 0,Y 213.709,Z 323.858,A -85,B 0,C 180,E1 -20743.678,E2 -20743.678} C_VEL
LIN {X 0,Y 213.709,Z 323.865,A -85,B 0,C 180,E1 -20746.344,E2 -20746.344} C_VEL
LIN {X 0,Y 213.709,Z 323.864,A -85,B 0,C 180,E1 -20751.326,E2 -20751.326} C_VEL
LIN {X 0,Y 213.755,Z 323.854,A -85,B 0,C 180,E1 -20756.013,E2 -20756.013} C_VEL
LIN {X 0,Y 213.749,Z 323.861,A -85,B 0,C 180,E1 -20760.444,E2 -20760.444} C_VEL
LIN {X 0,Y 213.788,Z 323.859,A -85,B 0,C 180,E1 -20764.695,E2 -20764.695} C_VEL
LIN {X 0,Y 213.787,Z 323.86,A -85,B 0,C 180,E1 -20768.796,E2 -20768.796} C_VEL
LIN {X 0,Y 213.893,Z 323.845,A -85,B 0,C 180,E1 -20772.794,E2 -20772.794} C_VEL
LIN {X 0,Y 213.94,Z 323.837,A -85,B 0,C 180,E1 -20776.7,E2 -20776.7} C_VEL
LIN {X 0,Y 214.139,Z 323.809,A -85,B 0,C 180,E1 -20780.55,E2 -20780.55} C_VEL
LIN {X 0,Y 214.077,Z 323.819,A -85,B 0,C 180,E1 -20784.342,E2 -20784.342} C_VEL
LIN {X 0,Y 214.174,Z 323.807,A -85,B 0,C 180,E1 -20786.761,E2 -20786.761} C_VEL
LIN {X 0,Y 215.221,Z 326.638,A -85,B 0,C 180,E1 -20787.061,E2 -20787.061} C_VEL
LIN {X 0,Y 217.935,Z 331.307,A -85,B 0,C 180,E1 -20787.644,E2 -20787.644} C_VEL
LIN {X 0,Y 223.439,Z 342.8,A -85,B 0,C 180,E1 -20788.872,E2 -20788.872} C_VEL
LIN {X 0,Y 230.857,Z 362.453,A -85,B 0,C 180,E1 -20790.573,E2 -20790.573} C_VEL
LIN {X 0,Y 231.428,Z 364.059,A -85,B 0,C 180,E1 -20790.702,E2 -20790.702} C_VEL
LIN {X 0,Y 228.56,Z 428.131,A -85,B 0,C 180,E1 -20792.806,E2 -20792.806} C_VEL
LIN {X 0,Y 227.423,Z 442.078,A -85,B 0,C 180,E1 -20793.636,E2 -20793.636} C_VEL
LIN {X 0,Y 226.027,Z 454.595,A -85,B 0,C 180,E1 -20794.748,E2 -20794.748} C_VEL
LIN {X 0,Y 224.095,Z 467.408,A -85,B 0,C 180,E1 -20796.295,E2 -20796.295} C_VEL
LIN {X 0,Y 222.162,Z 478.014,A -85,B 0,C 180,E1 -20797.949,E2 -20797.949} C_VEL
LIN {X 0,Y 220.017,Z 488.483,A -85,B 0,C 180,E1 -20800.019,E2 -20800.019} C_VEL
LIN {X 0,Y 217.852,Z 498.648,A -85,B 0,C 180,E1 -20802.57,E2 -20802.57} C_VEL
LIN {X 0,Y 216.058,Z 506.614,A -85,B 0,C 180,E1 -20805.076,E2 -20805.076} C_VEL
LIN {X 0,Y 214.371,Z 514.082,A -85,B 0,C 180,E1 -20808.057,E2 -20808.057} C_VEL
LIN {X 0,Y 213.078,Z 520.31,A -85,B 0,C 180,E1 -20811.265,E2 -20811.265} C_VEL
LIN {X 0,Y 212.185,Z 524.947,A -85,B 0,C 180,E1 -20814.449,E2 -20814.449} C_VEL
LIN {X 0,Y 211.46,Z 528.291,A -85,B 0,C 180,E1 -20817.721,E2 -20817.721} C_VEL
LIN {X 0,Y 211.21,Z 529.94,A -85,B 0,C 180,E1 -20820.1,E2 -20820.1} C_VEL
LIN {X 0,Y 211.228,Z 531.202,A -85,B 0,C 180,E1 -20823.715,E2 -20823.715} C_VEL
LIN {X 0,Y 211.713,Z 531.064,A -85,B 0,C 180,E1 -20827.183,E2 -20827.183} C_VEL
LIN {X 0,Y 212.58,Z 529.705,A -85,B 0,C 180,E1 -20830.501,E2 -20830.501} C_VEL
LIN {X 0,Y 213.937,Z 527.172,A -85,B 0,C 180,E1 -20833.72,E2 -20833.72} C_VEL
LIN {X 0,Y 215.572,Z 523.555,A -85,B 0,C 180,E1 -20836.793,E2 -20836.793} C_VEL
LIN {X 0,Y 217.718,Z 518.675,A -85,B 0,C 180,E1 -20839.789,E2 -20839.789} C_VEL
LIN {X 0,Y 220.554,Z 512.151,A -85,B 0,C 180,E1 -20842.795,E2 -20842.795} C_VEL
LIN {X 0,Y 223.73,Z 504.351,A -85,B 0,C 180,E1 -20845.567,E2 -20845.567} C_VEL
LIN {X 0,Y 226.9,Z 495.527,A -85,B 0,C 180,E1 -20848.015,E2 -20848.015} C_VEL
LIN {X 0,Y 229.949,Z 485.965,A -85,B 0,C 180,E1 -20850.12,E2 -20850.12} C_VEL
LIN {X 0,Y 233.038,Z 475.691,A -85,B 0,C 180,E1 -20851.88,E2 -20851.88} C_VEL
LIN {X 0,Y 235.733,Z 464.494,A -85,B 0,C 180,E1 -20853.411,E2 -20853.411} C_VEL
LIN {X 0,Y 238.239,Z 451.784,A -85,B 0,C 180,E1 -20854.715,E2 -20854.715} C_VEL
LIN {X 0,Y 240.052,Z 438.714,A -85,B 0,C 180,E1 -20855.701,E2 -20855.701} C_VEL
LIN {X 0,Y 241.443,Z 425.226,A -85,B 0,C 180,E1 -20856.313,E2 -20856.313} C_VEL
LIN {X 0,Y 244.416,Z 374.089,A -85,B 0,C 180,E1 -20857.926,E2 -20857.926} C_VEL
LIN {X 0,Y 239.303,Z 362.768,A -85,B 0,C 180,E1 -20859.617,E2 -20859.617} C_VEL
LIN {X 0,Y 233.927,Z 352.822,A -85,B 0,C 180,E1 -20861.476,E2 -20861.476} C_VEL
LIN {X 0,Y 229.249,Z 345.614,A -85,B 0,C 180,E1 -20863.167,E2 -20863.167} C_VEL
LIN {X 0,Y 226.726,Z 341.978,A -85,B 0,C 180,E1 -20864.134,E2 -20864.134} C_VEL
LIN {X 0,Y 224.099,Z 338.163,A -85,B 0,C 180,E1 -20865.193,E2 -20865.193} C_VEL
LIN {X 0,Y 221.682,Z 334.59,A -85,B 0,C 180,E1 -20866.245,E2 -20866.245} C_VEL
LIN {X 0,Y 218.843,Z 331.417,A -85,B 0,C 180,E1 -20867.48,E2 -20867.48} C_VEL
LIN {X 0,Y 217.558,Z 329.179,A -85,B 0,C 180,E1 -20868.115,E2 -20868.115} C_VEL
LIN {X 0,Y 215.312,Z 327.152,A -85,B 0,C 180,E1 -20869.144,E2 -20869.144} C_VEL
LIN {X 0,Y 214.206,Z 324.697,A -85,B 0,C 180,E1 -20869.773,E2 -20869.773} C_VEL
LIN {X 0,Y 214.08,Z 323.812,A -85,B 0,C 180,E1 -20869.962,E2 -20869.962} C_VEL
LIN {X 0,Y 214.152,Z 323.801,A -85,B 0,C 180,E1 -20872.457,E2 -20872.457} C_VEL
LIN {X 0,Y 214.404,Z 323.777,A -85,B 0,C 180,E1 -20878.121,E2 -20878.121} C_VEL
LIN {X 0,Y 214.505,Z 323.753,A -85,B 0,C 180,E1 -20880,E2 -20880} C_VEL
LIN {X 0,Y 214.405,Z 323.777,A -85,B 0,C 180,E1 -20881.878,E2 -20881.878} C_VEL
LIN {X 0,Y 214.166,Z 323.795,A -85,B 0,C 180,E1 -20887.543,E2 -20887.543} C_VEL
LIN {X 0,Y 213.974,Z 323.821,A -85,B 0,C 180,E1 -20891.366,E2 -20891.366} C_VEL
LIN {X 0,Y 213.885,Z 323.833,A -85,B 0,C 180,E1 -20895.24,E2 -20895.24} C_VEL
LIN {X 0,Y 213.847,Z 323.838,A -85,B 0,C 180,E1 -20899.187,E2 -20899.187} C_VEL
LIN {X 0,Y 213.828,Z 323.84,A -85,B 0,C 180,E1 -20903.229,E2 -20903.229} C_VEL
LIN {X 0,Y 213.798,Z 323.843,A -85,B 0,C 180,E1 -20907.454,E2 -20907.454} C_VEL
LIN {X 0,Y 213.74,Z 323.851,A -85,B 0,C 180,E1 -20911.742,E2 -20911.742} C_VEL
LIN {X 0,Y 213.749,Z 323.853,A -85,B 0,C 180,E1 -20914.847,E2 -20914.847} C_VEL
LIN {X 0,Y 213.074,Z 324.296,A -85,B 0,C 180,E1 -20915.923,E2 -20915.923} C_VEL
LIN {X 0,Y 211.664,Z 325.418,A -85,B 0,C 180,E1 -20916.936,E2 -20916.936} C_VEL
LIN {X 0,Y 209.38,Z 328.265,A -85,B 0,C 180,E1 -20918.533,E2 -20918.533} C_VEL
LIN {X 0,Y 209.027,Z 330.715,A -85,B 0,C 180,E1 -20919.631,E2 -20919.631} C_VEL
LIN {X 0,Y 209.497,Z 331.781,A -85,B 0,C 180,E1 -20920.076,E2 -20920.076} C_VEL
LIN {X 0,Y 213.623,Z 337.367,A -85,B 0,C 180,E1 -20922.336,E2 -20922.336} C_VEL
LIN {X 0,Y 216.969,Z 342.372,A -85,B 0,C 180,E1 -20923.994,E2 -20923.994} C_VEL
LIN {X 0,Y 221.457,Z 349.693,A -85,B 0,C 180,E1 -20926.077,E2 -20926.077} C_VEL
LIN {X 0,Y 227.129,Z 359.654,A -85,B 0,C 180,E1 -20928.443,E2 -20928.443} C_VEL
LIN {X 0,Y 232.399,Z 370.563,A -85,B 0,C 180,E1 -20930.485,E2 -20930.485} C_VEL
LIN {X 0,Y 236.9,Z 381.452,A -85,B 0,C 180,E1 -20932.164,E2 -20932.164} C_VEL
LIN {X 0,Y 238.198,Z 393.822,A -85,B 0,C 180,E1 -20933.042,E2 -20933.042} C_VEL
LIN {X 0,Y 235.178,Z 442.248,A -85,B 0,C 180,E1 -20934.625,E2 -20934.625} C_VEL
LIN {X 0,Y 233.505,Z 455.41,A -85,B 0,C 180,E1 -20935.326,E2 -20935.326} C_VEL
LIN {X 0,Y 231.126,Z 468.109,A -85,B 0,C 180,E1 -20936.303,E2 -20936.303} C_VEL
LIN {X 0,Y 228.129,Z 480.556,A -85,B 0,C 180,E1 -20937.647,E2 -20937.647} C_VEL
LIN {X 0,Y 224.987,Z 491.712,A -85,B 0,C 180,E1 -20939.245,E2 -20939.245} C_VEL
LIN {X 0,Y 221.673,Z 501.861,A -85,B 0,C 180,E1 -20941.095,E2 -20941.095} C_VEL
LIN {X 0,Y 218.4,Z 511.032,A -85,B 0,C 180,E1 -20943.232,E2 -20943.232} C_VEL
LIN {X 0,Y 214.86,Z 520.031,A -85,B 0,C 180,E1 -20945.875,E2 -20945.875} C_VEL
LIN {X 0,Y 211.968,Z 527.319,A -85,B 0,C 180,E1 -20948.618,E2 -20948.618} C_VEL
LIN {X 0,Y 209.467,Z 533.195,A -85,B 0,C 180,E1 -20951.421,E2 -20951.421} C_VEL
LIN {X 0,Y 207.364,Z 537.857,A -85,B 0,C 180,E1 -20954.276,E2 -20954.276} C_VEL
LIN {X 0,Y 205.938,Z 541.436,A -85,B 0,C 180,E1 -20957.191,E2 -20957.191} C_VEL
LIN {X 0,Y 205.011,Z 544.028,A -85,B 0,C 180,E1 -20960.138,E2 -20960.138} C_VEL
LIN {X 0,Y 204.621,Z 545.261,A -85,B 0,C 180,E1 -20962.11,E2 -20962.11} C_VEL
LIN {X 0,Y 204.335,Z 546.473,A -85,B 0,C 180,E1 -20966.062,E2 -20966.062} C_VEL
LIN {X 0,Y 204.437,Z 546.5,A -85,B 0,C 180,E1 -20968.036,E2 -20968.036} C_VEL
LIN {X 0,Y 204.575,Z 546.129,A -85,B 0,C 180,E1 -20970.006,E2 -20970.006} C_VEL
LIN {X 0,Y 204.477,Z 545.297,A -85,B 0,C 180,E1 -20971.976,E2 -20971.976} C_VEL
LIN {X 0,Y 204.413,Z 543.72,A -85,B 0,C 180,E1 -20974.393,E2 -20974.393} C_VEL
LIN {X 0,Y 204.649,Z 540.25,A -85,B 0,C 180,E1 -20977.901,E2 -20977.901} C_VEL
LIN {X 0,Y 205.175,Z 536.122,A -85,B 0,C 180,E1 -20980.865,E2 -20980.865} C_VEL
LIN {X 0,Y 206.365,Z 529.762,A -85,B 0,C 180,E1 -20984.3,E2 -20984.3} C_VEL
LIN {X 0,Y 207.891,Z 522.813,A -85,B 0,C 180,E1 -20987.211,E2 -20987.211} C_VEL
LIN {X 0,Y 209.566,Z 515.707,A -85,B 0,C 180,E1 -20989.6,E2 -20989.6} C_VEL
LIN {X 0,Y 211.492,Z 507.108,A -85,B 0,C 180,E1 -20991.958,E2 -20991.958} C_VEL
LIN {X 0,Y 213.541,Z 497.658,A -85,B 0,C 180,E1 -20994.039,E2 -20994.039} C_VEL
LIN {X 0,Y 215.94,Z 485.966,A -85,B 0,C 180,E1 -20996.069,E2 -20996.069} C_VEL
LIN {X 0,Y 217.73,Z 476.233,A -85,B 0,C 180,E1 -20997.39,E2 -20997.39} C_VEL
LIN {X 0,Y 219.606,Z 463.823,A -85,B 0,C 180,E1 -20998.693,E2 -20998.693} C_VEL
LIN {X 0,Y 221.135,Z 450.788,A -85,B 0,C 180,E1 -20999.648,E2 -20999.648} C_VEL
LIN {X 0,Y 222.134,Z 437.144,A -85,B 0,C 180,E1 -21000.285,E2 -21000.285} C_VEL
LIN {X 0,Y 224.054,Z 390.266,A -85,B 0,C 180,E1 -21001.853,E2 -21001.853} C_VEL
LIN {X 0,Y 220.847,Z 364.192,A -85,B 0,C 180,E1 -21003.285,E2 -21003.285} C_VEL
LIN {X 0,Y 213.028,Z 344.047,A -85,B 0,C 180,E1 -21005.197,E2 -21005.197} C_VEL
LIN {X 0,Y 208.926,Z 334.126,A -85,B 0,C 180,E1 -21006.287,E2 -21006.287} C_VEL
LIN {X 0,Y 207.025,Z 326.095,A -85,B 0,C 180,E1 -21010.171,E2 -21010.171} C_VEL
LIN {X 0,Y 206.701,Z 324.745,A -85,B 0,C 180,E1 -21010.931,E2 -21010.931} C_VEL
LIN {X 0,Y 206.64,Z 324.75,A -85,B 0,C 180,E1 -21015.585,E2 -21015.585} C_VEL
LIN {X 0,Y 206.66,Z 324.742,A -85,B 0,C 180,E1 -21019.748,E2 -21019.748} C_VEL
LIN {X 0,Y 206.709,Z 324.736,A -85,B 0,C 180,E1 -21024.691,E2 -21024.691} C_VEL
LIN {X 0,Y 206.715,Z 324.732,A -85,B 0,C 180,E1 -21029.338,E2 -21029.338} C_VEL
LIN {X 0,Y 206.738,Z 324.73,A -85,B 0,C 180,E1 -21033.773,E2 -21033.773} C_VEL
LIN {X 0,Y 206.724,Z 324.733,A -85,B 0,C 180,E1 -21038.04,E2 -21038.04} C_VEL
LIN {X 0,Y 206.812,Z 324.702,A -85,B 0,C 180,E1 -21042.191,E2 -21042.191} C_VEL
LIN {X 0,Y 206.878,Z 324.702,A -85,B 0,C 180,E1 -21046.243,E2 -21046.243} C_VEL
LIN {X 0,Y 207.081,Z 324.688,A -85,B 0,C 180,E1 -21050.23,E2 -21050.23} C_VEL
LIN {X 0,Y 207.059,Z 324.679,A -85,B 0,C 180,E1 -21054.156,E2 -21054.156} C_VEL
LIN {X 0,Y 207.365,Z 324.615,A -85,B 0,C 180,E1 -21058.058,E2 -21058.058} C_VEL
LIN {X 0,Y 207.508,Z 324.609,A -85,B 0,C 180,E1 -21060,E2 -21060} C_VEL
LIN {X 0,Y 207.38,Z 324.641,A -85,B 0,C 180,E1 -21061.942,E2 -21061.942} C_VEL
LIN {X 0,Y 207.122,Z 324.682,A -85,B 0,C 180,E1 -21067.801,E2 -21067.801} C_VEL
LIN {X 0,Y 206.914,Z 324.704,A -85,B 0,C 180,E1 -21071.759,E2 -21071.759} C_VEL
LIN {X 0,Y 206.82,Z 324.722,A -85,B 0,C 180,E1 -21075.774,E2 -21075.774} C_VEL
LIN {X 0,Y 206.719,Z 324.724,A -85,B 0,C 180,E1 -21079.876,E2 -21079.876} C_VEL
LIN {X 0,Y 206.705,Z 324.736,A -85,B 0,C 180,E1 -21084.08,E2 -21084.08} C_VEL
LIN {X 0,Y 206.678,Z 324.718,A -85,B 0,C 180,E1 -21088.429,E2 -21088.429} C_VEL
LIN {X 0,Y 206.684,Z 324.707,A -85,B 0,C 180,E1 -21092.961,E2 -21092.961} C_VEL
LIN {X 0,Y 206.709,Z 324.725,A -85,B 0,C 180,E1 -21095.31,E2 -21095.31} C_VEL
LIN {X 0,Y 206.652,Z 324.744,A -85,B 0,C 180,E1 -21100.254,E2 -21100.254} C_VEL
LIN {X 0,Y 206.637,Z 324.742,A -85,B 0,C 180,E1 -21104.414,E2 -21104.414} C_VEL
LIN {X 0,Y 206.636,Z 324.742,A -85,B 0,C 180,E1 -21108.44,E2 -21108.44} C_VEL
LIN {X 0,Y 206.672,Z 324.741,A -85,B 0,C 180,E1 -21112.254,E2 -21112.254} C_VEL
LIN {X 0,Y 206.709,Z 324.734,A -85,B 0,C 180,E1 -21114.686,E2 -21114.686} C_VEL
LIN {X 0,Y 206.7,Z 324.739,A -85,B 0,C 180,E1 -21119.33,E2 -21119.33} C_VEL
LIN {X 0,Y 206.711,Z 324.74,A -85,B 0,C 180,E1 -21123.764,E2 -21123.764} C_VEL
LIN {X 0,Y 206.726,Z 324.738,A -85,B 0,C 180,E1 -21128.034,E2 -21128.034} C_VEL
LIN {X 0,Y 206.829,Z 324.724,A -85,B 0,C 180,E1 -21132.187,E2 -21132.187} C_VEL
LIN {X 0,Y 206.881,Z 324.716,A -85,B 0,C 180,E1 -21136.238,E2 -21136.238} C_VEL
LIN {X 0,Y 207.084,Z 324.688,A -85,B 0,C 180,E1 -21140.224,E2 -21140.224} C_VEL
LIN {X 0,Y 207.041,Z 324.696,A -85,B 0,C 180,E1 -21144.149,E2 -21144.149} C_VEL
LIN {X 0,Y 207.031,Z 324.692,A -85,B 0,C 180,E1 -21145.674,E2 -21145.674} C_VEL
LIN {X 0,Y 208.237,Z 327.811,A -85,B 0,C 180,E1 -21146.046,E2 -21146.046} C_VEL
LIN {X 0,Y 213.691,Z 337.508,A -85,B 0,C 180,E1 -21147.287,E2 -21147.287} C_VEL
LIN {X 0,Y 217.967,Z 346.86,A -85,B 0,C 180,E1 -21148.278,E2 -21148.278} C_VEL
LIN {X 0,Y 224.778,Z 365.016,A -85,B 0,C 180,E1 -21149.91,E2 -21149.91} C_VEL
LIN {X 0,Y 224.849,Z 369.757,A -85,B 0,C 180,E1 -21150.102,E2 -21150.102} C_VEL
LIN {X 0,Y 222.12,Z 427.519,A -85,B 0,C 180,E1 -21152.034,E2 -21152.034} C_VEL
LIN {X 0,Y 221.007,Z 441.136,A -85,B 0,C 180,E1 -21152.842,E2 -21152.842} C_VEL
LIN {X 0,Y 219.57,Z 454.013,A -85,B 0,C 180,E1 -21153.981,E2 -21153.981} C_VEL
LIN {X 0,Y 217.913,Z 465.099,A -85,B 0,C 180,E1 -21155.303,E2 -21155.303} C_VEL
LIN {X 0,Y 215.821,Z 476.258,A -85,B 0,C 180,E1 -21157.008,E2 -21157.008} C_VEL
LIN {X 0,Y 213.551,Z 487.205,A -85,B 0,C 180,E1 -21159.137,E2 -21159.137} C_VEL
LIN {X 0,Y 211.437,Z 496.741,A -85,B 0,C 180,E1 -21161.497,E2 -21161.497} C_VEL
LIN {X 0,Y 209.576,Z 504.898,A -85,B 0,C 180,E1 -21164.014,E2 -21164.014} C_VEL
LIN {X 0,Y 207.947,Z 511.897,A -85,B 0,C 180,E1 -21166.687,E2 -21166.687} C_VEL
LIN {X 0,Y 206.448,Z 518.54,A -85,B 0,C 180,E1 -21169.895,E2 -21169.895} C_VEL
LIN {X 0,Y 205.39,Z 523.888,A -85,B 0,C 180,E1 -21173.351,E2 -21173.351} C_VEL
LIN {X 0,Y 204.547,Z 527.64,A -85,B 0,C 180,E1 -21176.705,E2 -21176.705} C_VEL
LIN {X 0,Y 204.214,Z 529.341,A -85,B 0,C 180,E1 -21178.794,E2 -21178.794} C_VEL
LIN {X 0,Y 204.056,Z 530.617,A -85,B 0,C 180,E1 -21181.096,E2 -21181.096} C_VEL
LIN {X 0,Y 204.217,Z 531.509,A -85,B 0,C 180,E1 -21184.315,E2 -21184.315} C_VEL
LIN {X 0,Y 204.816,Z 531.214,A -85,B 0,C 180,E1 -21188.133,E2 -21188.133} C_VEL
LIN {X 0,Y 205.742,Z 529.829,A -85,B 0,C 180,E1 -21191.279,E2 -21191.279} C_VEL
LIN {X 0,Y 207.208,Z 527.224,A -85,B 0,C 180,E1 -21194.58,E2 -21194.58} C_VEL
LIN {X 0,Y 209.028,Z 523.489,A -85,B 0,C 180,E1 -21197.744,E2 -21197.744} C_VEL
LIN {X 0,Y 211.424,Z 518.467,A -85,B 0,C 180,E1 -21200.833,E2 -21200.833} C_VEL
LIN {X 0,Y 214.384,Z 512.008,A -85,B 0,C 180,E1 -21203.837,E2 -21203.837} C_VEL
LIN {X 0,Y 217.241,Z 505.348,A -85,B 0,C 180,E1 -21206.262,E2 -21206.262} C_VEL
LIN {X 0,Y 220.675,Z 496.47,A -85,B 0,C 180,E1 -21208.842,E2 -21208.842} C_VEL
LIN {X 0,Y 223.941,Z 486.82,A -85,B 0,C 180,E1 -21211.045,E2 -21211.045} C_VEL
LIN {X 0,Y 227.39,Z 475.931,A -85,B 0,C 180,E1 -21212.958,E2 -21212.958} C_VEL
LIN {X 0,Y 230.303,Z 464.339,A -85,B 0,C 180,E1 -21214.554,E2 -21214.554} C_VEL
LIN {X 0,Y 232.911,Z 451.563,A -85,B 0,C 180,E1 -21215.87,E2 -21215.87} C_VEL
LIN {X 0,Y 234.766,Z 438.614,A -85,B 0,C 180,E1 -21216.844,E2 -21216.844} C_VEL
LIN {X 0,Y 236.197,Z 424.959,A -85,B 0,C 180,E1 -21217.464,E2 -21217.464} C_VEL
LIN {X 0,Y 239.154,Z 376.456,A -85,B 0,C 180,E1 -21219.013,E2 -21219.013} C_VEL
LIN {X 0,Y 233.9,Z 364.84,A -85,B 0,C 180,E1 -21220.888,E2 -21220.888} C_VEL
LIN {X 0,Y 228.778,Z 355.609,A -85,B 0,C 180,E1 -21222.77,E2 -21222.77} C_VEL
LIN {X 0,Y 223.043,Z 347.022,A -85,B 0,C 180,E1 -21225.03,E2 -21225.03} C_VEL
LIN {X 0,Y 220.532,Z 343.38,A -85,B 0,C 180,E1 -21226.113,E2 -21226.113} C_VEL
LIN {X 0,Y 217.983,Z 339.783,A -85,B 0,C 180,E1 -21227.267,E2 -21227.267} C_VEL
LIN {X 0,Y 215.403,Z 336.376,A -85,B 0,C 180,E1 -21228.487,E2 -21228.487} C_VEL
LIN {X 0,Y 214.486,Z 335.127,A -85,B 0,C 180,E1 -21228.941,E2 -21228.941} C_VEL
LIN {X 0,Y 212.091,Z 332.312,A -85,B 0,C 180,E1 -21230.159,E2 -21230.159} C_VEL
LIN {X 0,Y 211.065,Z 330.237,A -85,B 0,C 180,E1 -21230.779,E2 -21230.779} C_VEL
LIN {X 0,Y 208.678,Z 328.362,A -85,B 0,C 180,E1 -21232.075,E2 -21232.075} C_VEL
LIN {X 0,Y 207.281,Z 325.734,A -85,B 0,C 180,E1 -21233.001,E2 -21233.001} C_VEL
LIN {X 0,Y 207.052,Z 324.686,A -85,B 0,C 180,E1 -21233.299,E2 -21233.299} C_VEL
LIN {X 0,Y 207.34,Z 324.658,A -85,B 0,C 180,E1 -21238.057,E2 -21238.057} C_VEL
LIN {X 0,Y 207.471,Z 324.629,A -85,B 0,C 180,E1 -21240,E2 -21240} C_VEL
LIN {X 0,Y 207.342,Z 324.657,A -85,B 0,C 180,E1 -21241.942,E2 -21241.942} C_VEL
LIN {X 0,Y 207.109,Z 324.674,A -85,B 0,C 180,E1 -21247.801,E2 -21247.801} C_VEL
LIN {X 0,Y 206.895,Z 324.7,A -85,B 0,C 180,E1 -21251.76,E2 -21251.76} C_VEL
LIN {X 0,Y 206.821,Z 324.709,A -85,B 0,C 180,E1 -21255.774,E2 -21255.774} C_VEL
LIN {X 0,Y 206.786,Z 324.712,A -85,B 0,C 180,E1 -21259.869,E2 -21259.869} C_VEL
LIN {X 0,Y 206.739,Z 324.718,A -85,B 0,C 180,E1 -21264.075,E2 -21264.075} C_VEL
LIN {X 0,Y 206.713,Z 324.723,A -85,B 0,C 180,E1 -21268.423,E2 -21268.423} C_VEL
LIN {X 0,Y 206.677,Z 324.735,A -85,B 0,C 180,E1 -21272.962,E2 -21272.962} C_VEL
LIN {X 0,Y 206.74,Z 324.889,A -85,B 0,C 180,E1 -21274.709,E2 -21274.709} C_VEL
LIN {X 0,Y 208.656,Z 330.165,A -85,B 0,C 180,E1 -21279.531,E2 -21279.531} C_VEL
LIN {X 0,Y 209.497,Z 331.781,A -85,B 0,C 180,E1 -21280.076,E2 -21280.076} C_VEL
LIN {X 0,Y 211.392,Z 335.418,A -85,B 0,C 180,E1 -21281.233,E2 -21281.233} C_VEL
LIN {X 0,Y 213.885,Z 342.978,A -85,B 0,C 180,E1 -21282.825,E2 -21282.825} C_VEL
LIN {X 0,Y 216.911,Z 352.483,A -85,B 0,C 180,E1 -21284.622,E2 -21284.622} C_VEL
LIN {X 0,Y 218.238,Z 355.296,A -85,B 0,C 180,E1 -21285.285,E2 -21285.285} C_VEL
LIN {X 0,Y 223.365,Z 364.567,A -85,B 0,C 180,E1 -21287.554,E2 -21287.554} C_VEL
LIN {X 0,Y 228.484,Z 375.553,A -85,B 0,C 180,E1 -21289.674,E2 -21289.674} C_VEL
LIN {X 0,Y 232.194,Z 385.04,A -85,B 0,C 180,E1 -21291.148,E2 -21291.148} C_VEL
LIN {X 0,Y 233.121,Z 395.424,A -85,B 0,C 180,E1 -21291.893,E2 -21291.893} C_VEL
LIN {X 0,Y 229.925,Z 442.427,A -85,B 0,C 180,E1 -21293.448,E2 -21293.448} C_VEL
LIN {X 0,Y 228.122,Z 455.808,A -85,B 0,C 180,E1 -21294.182,E2 -21294.182} C_VEL
LIN {X 0,Y 225.748,Z 467.798,A -85,B 0,C 180,E1 -21295.116,E2 -21295.116} C_VEL
LIN {X 0,Y 222.66,Z 480.247,A -85,B 0,C 180,E1 -21296.48,E2 -21296.48} C_VEL
LIN {X 0,Y 219.378,Z 491.411,A -85,B 0,C 180,E1 -21298.099,E2 -21298.099} C_VEL
LIN {X 0,Y 215.897,Z 501.569,A -85,B 0,C 180,E1 -21299.976,E2 -21299.976} C_VEL
LIN {X 0,Y 212.109,Z 511.558,A -85,B 0,C 180,E1 -21302.372,E2 -21302.372} C_VEL
LIN {X 0,Y 208.421,Z 520.401,A -85,B 0,C 180,E1 -21305.079,E2 -21305.079} C_VEL
LIN {X 0,Y 205.381,Z 527.543,A -85,B 0,C 180,E1 -21307.897,E2 -21307.897} C_VEL
LIN {X 0,Y 202.742,Z 533.296,A -85,B 0,C 180,E1 -21310.781,E2 -21310.781} C_VEL
LIN {X 0,Y 200.537,Z 537.875,A -85,B 0,C 180,E1 -21313.726,E2 -21313.726} C_VEL
LIN {X 0,Y 198.996,Z 541.39,A -85,B 0,C 180,E1 -21316.736,E2 -21316.736} C_VEL
LIN {X 0,Y 197.988,Z 543.921,A -85,B 0,C 180,E1 -21319.784,E2 -21319.784} C_VEL
LIN {X 0,Y 197.571,Z 545.084,A -85,B 0,C 180,E1 -21321.827,E2 -21321.827} C_VEL
LIN {X 0,Y 197.247,Z 546.222,A -85,B 0,C 180,E1 -21325.921,E2 -21325.921} C_VEL
LIN {X 0,Y 197.336,Z 546.215,A -85,B 0,C 180,E1 -21327.966,E2 -21327.966} C_VEL
LIN {X 0,Y 197.489,Z 545.789,A -85,B 0,C 180,E1 -21330.007,E2 -21330.007} C_VEL
LIN {X 0,Y 197.376,Z 544.916,A -85,B 0,C 180,E1 -21332.047,E2 -21332.047} C_VEL
LIN {X 0,Y 197.345,Z 543.47,A -85,B 0,C 180,E1 -21334.32,E2 -21334.32} C_VEL
LIN {X 0,Y 197.461,Z 540.871,A -85,B 0,C 180,E1 -21337.162,E2 -21337.162} C_VEL
LIN {X 0,Y 197.943,Z 537.046,A -85,B 0,C 180,E1 -21340.232,E2 -21340.232} C_VEL
LIN {X 0,Y 198.798,Z 532.051,A -85,B 0,C 180,E1 -21343.291,E2 -21343.291} C_VEL
LIN {X 0,Y 200.228,Z 525.75,A -85,B 0,C 180,E1 -21346.314,E2 -21346.314} C_VEL
LIN {X 0,Y 201.792,Z 519.285,A -85,B 0,C 180,E1 -21348.799,E2 -21348.799} C_VEL
LIN {X 0,Y 203.553,Z 511.636,A -85,B 0,C 180,E1 -21351.216,E2 -21351.216} C_VEL
LIN {X 0,Y 205.716,Z 501.985,A -85,B 0,C 180,E1 -21353.672,E2 -21353.672} C_VEL
LIN {X 0,Y 207.846,Z 492.753,A -85,B 0,C 180,E1 -21355.544,E2 -21355.544} C_VEL
LIN {X 0,Y 210.234,Z 481.368,A -85,B 0,C 180,E1 -21357.37,E2 -21357.37} C_VEL
LIN {X 0,Y 212.081,Z 470.555,A -85,B 0,C 180,E1 -21358.723,E2 -21358.723} C_VEL
LIN {X 0,Y 213.716,Z 458.86,A -85,B 0,C 180,E1 -21359.832,E2 -21359.832} C_VEL
LIN {X 0,Y 215.036,Z 446.446,A -85,B 0,C 180,E1 -21360.645,E2 -21360.645} C_VEL
LIN {X 0,Y 215.983,Z 429.725,A -85,B 0,C 180,E1 -21361.311,E2 -21361.311} C_VEL
LIN {X 0,Y 217.676,Z 391.074,A -85,B 0,C 180,E1 -21362.635,E2 -21362.635} C_VEL
LIN {X 0,Y 214.704,Z 366.489,A -85,B 0,C 180,E1 -21364.032,E2 -21364.032} C_VEL
LIN {X 0,Y 206.413,Z 345.058,A -85,B 0,C 180,E1 -21366.152,E2 -21366.152} C_VEL
LIN {X 0,Y 201.651,Z 333.93,A -85,B 0,C 180,E1 -21367.425,E2 -21367.425} C_VEL
LIN {X 0,Y 199.604,Z 325.624,A -85,B 0,C 180,E1 -21371.732,E2 -21371.732} C_VEL
LIN {X 0,Y 199.586,Z 325.629,A -85,B 0,C 180,E1 -21375.23,E2 -21375.23} C_VEL
LIN {X 0,Y 199.583,Z 325.626,A -85,B 0,C 180,E1 -21378.006,E2 -21378.006} C_VEL
LIN {X 0,Y 199.607,Z 325.622,A -85,B 0,C 180,E1 -21380.775,E2 -21380.775} C_VEL
LIN {X 0,Y 199.62,Z 325.618,A -85,B 0,C 180,E1 -21385.715,E2 -21385.715} C_VEL
LIN {X 0,Y 199.701,Z 325.612,A -85,B 0,C 180,E1 -21388.137,E2 -21388.137} C_VEL
LIN {X 0,Y 199.694,Z 325.612,A -85,B 0,C 180,E1 -21392.773,E2 -21392.773} C_VEL
LIN {X 0,Y 199.688,Z 325.612,A -85,B 0,C 180,E1 -21397.223,E2 -21397.223} C_VEL
LIN {X 0,Y 199.755,Z 325.584,A -85,B 0,C 180,E1 -21401.804,E2 -21401.804} C_VEL
LIN {X 0,Y 199.816,Z 325.576,A -85,B 0,C 180,E1 -21405.747,E2 -21405.747} C_VEL
LIN {X 0,Y 200.032,Z 325.567,A -85,B 0,C 180,E1 -21409.882,E2 -21409.882} C_VEL
LIN {X 0,Y 200.021,Z 325.556,A -85,B 0,C 180,E1 -21413.949,E2 -21413.949} C_VEL
LIN {X 0,Y 200.307,Z 325.492,A -85,B 0,C 180,E1 -21417.989,E2 -21417.989} C_VEL
LIN {X 0,Y 200.473,Z 325.483,A -85,B 0,C 180,E1 -21420,E2 -21420} C_VEL
LIN {X 0,Y 200.014,Z 325.569,A -85,B 0,C 180,E1 -21424.03,E2 -21424.03} C_VEL
LIN {X 0,Y 200.072,Z 325.558,A -85,B 0,C 180,E1 -21428.077,E2 -21428.077} C_VEL
LIN {X 0,Y 199.865,Z 325.585,A -85,B 0,C 180,E1 -21432.18,E2 -21432.18} C_VEL
LIN {X 0,Y 199.757,Z 325.598,A -85,B 0,C 180,E1 -21436.348,E2 -21436.348} C_VEL
LIN {X 0,Y 199.65,Z 325.61,A -85,B 0,C 180,E1 -21440.611,E2 -21440.611} C_VEL
LIN {X 0,Y 199.627,Z 325.614,A -85,B 0,C 180,E1 -21444.991,E2 -21444.991} C_VEL
LIN {X 0,Y 199.592,Z 325.589,A -85,B 0,C 180,E1 -21449.536,E2 -21449.536} C_VEL
LIN {X 0,Y 199.645,Z 325.575,A -85,B 0,C 180,E1 -21452.337,E2 -21452.337} C_VEL
LIN {X 0,Y 199.624,Z 325.615,A -85,B 0,C 180,E1 -21456.763,E2 -21456.763} C_VEL
LIN {X 0,Y 199.602,Z 325.62,A -85,B 0,C 180,E1 -21459.33,E2 -21459.33} C_VEL
LIN {X 0,Y 199.572,Z 325.618,A -85,B 0,C 180,E1 -21462.304,E2 -21462.304} C_VEL
LIN {X 0,Y 199.584,Z 325.623,A -85,B 0,C 180,E1 -21465.224,E2 -21465.224} C_VEL
LIN {X 0,Y 199.576,Z 325.623,A -85,B 0,C 180,E1 -21467.999,E2 -21467.999} C_VEL
LIN {X 0,Y 199.604,Z 325.618,A -85,B 0,C 180,E1 -21470.77,E2 -21470.77} C_VEL
LIN {X 0,Y 199.617,Z 325.615,A -85,B 0,C 180,E1 -21475.709,E2 -21475.709} C_VEL
LIN {X 0,Y 199.69,Z 325.612,A -85,B 0,C 180,E1 -21478.13,E2 -21478.13} C_VEL
LIN {X 0,Y 199.649,Z 325.618,A -85,B 0,C 180,E1 -21482.761,E2 -21482.761} C_VEL
LIN {X 0,Y 199.686,Z 325.614,A -85,B 0,C 180,E1 -21487.217,E2 -21487.217} C_VEL
LIN {X 0,Y 199.753,Z 325.606,A -85,B 0,C 180,E1 -21491.798,E2 -21491.798} C_VEL
LIN {X 0,Y 199.818,Z 325.597,A -85,B 0,C 180,E1 -21495.741,E2 -21495.741} C_VEL
LIN {X 0,Y 200.028,Z 325.568,A -85,B 0,C 180,E1 -21499.876,E2 -21499.876} C_VEL
LIN {X 0,Y 200.005,Z 325.573,A -85,B 0,C 180,E1 -21503.943,E2 -21503.943} C_VEL
LIN {X 0,Y 200.001,Z 325.571,A -85,B 0,C 180,E1 -21504.574,E2 -21504.574} C_VEL
LIN {X 0,Y 201.053,Z 328.498,A -85,B 0,C 180,E1 -21504.896,E2 -21504.896} C_VEL
LIN {X 0,Y 208.257,Z 341.392,A -85,B 0,C 180,E1 -21506.634,E2 -21506.634} C_VEL
LIN {X 0,Y 212.142,Z 349.89,A -85,B 0,C 180,E1 -21507.577,E2 -21507.577} C_VEL
LIN {X 0,Y 218.517,Z 366.912,A -85,B 0,C 180,E1 -21509.159,E2 -21509.159} C_VEL
LIN {X 0,Y 216.213,Z 417.773,A -85,B 0,C 180,E1 -21510.887,E2 -21510.887} C_VEL
LIN {X 0,Y 215.351,Z 432.195,A -85,B 0,C 180,E1 -21511.485,E2 -21511.485} C_VEL
LIN {X 0,Y 214.225,Z 444.573,A -85,B 0,C 180,E1 -21512.344,E2 -21512.344} C_VEL
LIN {X 0,Y 212.501,Z 457.871,A -85,B 0,C 180,E1 -21513.668,E2 -21513.668} C_VEL
LIN {X 0,Y 210.552,Z 469.454,A -85,B 0,C 180,E1 -21515.205,E2 -21515.205} C_VEL
LIN {X 0,Y 208.423,Z 480.023,A -85,B 0,C 180,E1 -21517.014,E2 -21517.014} C_VEL
LIN {X 0,Y 206.095,Z 490.511,A -85,B 0,C 180,E1 -21519.286,E2 -21519.286} C_VEL
LIN {X 0,Y 203.854,Z 500.172,A -85,B 0,C 180,E1 -21521.931,E2 -21521.931} C_VEL
LIN {X 0,Y 201.997,Z 507.911,A -85,B 0,C 180,E1 -21524.603,E2 -21524.603} C_VEL
LIN {X 0,Y 200.183,Z 515.332,A -85,B 0,C 180,E1 -21527.834,E2 -21527.834} C_VEL
LIN {X 0,Y 199.023,Z 520.446,A -85,B 0,C 180,E1 -21530.67,E2 -21530.67} C_VEL
LIN {X 0,Y 198.071,Z 525.183,A -85,B 0,C 180,E1 -21534.073,E2 -21534.073} C_VEL
LIN {X 0,Y 197.281,Z 528.641,A -85,B 0,C 180,E1 -21537.579,E2 -21537.579} C_VEL
LIN {X 0,Y 196.973,Z 530.807,A -85,B 0,C 180,E1 -21541.094,E2 -21541.094} C_VEL
LIN {X 0,Y 197.173,Z 531.814,A -85,B 0,C 180,E1 -21544.934,E2 -21544.934} C_VEL
LIN {X 0,Y 197.815,Z 531.487,A -85,B 0,C 180,E1 -21548.59,E2 -21548.59} C_VEL
LIN {X 0,Y 198.97,Z 529.925,A -85,B 0,C 180,E1 -21552.141,E2 -21552.141} C_VEL
LIN {X 0,Y 200.541,Z 527.241,A -85,B 0,C 180,E1 -21555.5,E2 -21555.5} C_VEL
LIN {X 0,Y 202.551,Z 523.41,A -85,B 0,C 180,E1 -21558.757,E2 -21558.757} C_VEL
LIN {X 0,Y 205.198,Z 518.245,A -85,B 0,C 180,E1 -21561.96,E2 -21561.96} C_VEL
LIN {X 0,Y 208.386,Z 511.729,A -85,B 0,C 180,E1 -21565.016,E2 -21565.016} C_VEL
LIN {X 0,Y 212.032,Z 503.472,A -85,B 0,C 180,E1 -21567.972,E2 -21567.972} C_VEL
LIN {X 0,Y 215.748,Z 494.057,A -85,B 0,C 180,E1 -21570.586,E2 -21570.586} C_VEL
LIN {X 0,Y 218.844,Z 485.329,A -85,B 0,C 180,E1 -21572.497,E2 -21572.497} C_VEL
LIN {X 0,Y 222.282,Z 474.529,A -85,B 0,C 180,E1 -21574.345,E2 -21574.345} C_VEL
LIN {X 0,Y 225.271,Z 462.871,A -85,B 0,C 180,E1 -21575.908,E2 -21575.908} C_VEL
LIN {X 0,Y 227.752,Z 450.95,A -85,B 0,C 180,E1 -21577.121,E2 -21577.121} C_VEL
LIN {X 0,Y 229.668,Z 437.877,A -85,B 0,C 180,E1 -21578.086,E2 -21578.086} C_VEL
LIN {X 0,Y 231.091,Z 424.742,A -85,B 0,C 180,E1 -21578.67,E2 -21578.67} C_VEL
LIN {X 0,Y 233.994,Z 378.789,A -85,B 0,C 180,E1 -21580.176,E2 -21580.176} C_VEL
LIN {X 0,Y 228.858,Z 367.574,A -85,B 0,C 180,E1 -21582.116,E2 -21582.116} C_VEL
LIN {X 0,Y 224.524,Z 359.872,A -85,B 0,C 180,E1 -21583.83,E2 -21583.83} C_VEL
LIN {X 0,Y 219.38,Z 351.952,A -85,B 0,C 180,E1 -21585.994,E2 -21585.994} C_VEL
LIN {X 0,Y 215.317,Z 345.944,A -85,B 0,C 180,E1 -21587.888,E2 -21587.888} C_VEL
LIN {X 0,Y 212.444,Z 342.077,A -85,B 0,C 180,E1 -21589.307,E2 -21589.307} C_VEL
LIN {X 0,Y 209.276,Z 337.964,A -85,B 0,C 180,E1 -21591.031,E2 -21591.031} C_VEL
LIN {X 0,Y 208.459,Z 336.543,A -85,B 0,C 180,E1 -21591.534,E2 -21591.534} C_VEL
LIN {X 0,Y 206.002,Z 334.132,A -85,B 0,C 180,E1 -21592.97,E2 -21592.97} C_VEL
LIN {X 0,Y 204.392,Z 331.289,A -85,B 0,C 180,E1 -21594.079,E2 -21594.079} C_VEL
LIN {X 0,Y 201.811,Z 329.497,A -85,B 0,C 180,E1 -21595.756,E2 -21595.756} C_VEL
LIN {X 0,Y 200.493,Z 327.175,A -85,B 0,C 180,E1 -21596.86,E2 -21596.86} C_VEL
LIN {X 0,Y 200.153,Z 325.548,A -85,B 0,C 180,E1 -21597.358,E2 -21597.358} C_VEL
LIN {X 0,Y 200.436,Z 325.505,A -85,B 0,C 180,E1 -21600,E2 -21600} C_VEL
LIN {X 0,Y 199.987,Z 325.561,A -85,B 0,C 180,E1 -21604.03,E2 -21604.03} C_VEL
LIN {X 0,Y 200.057,Z 325.552,A -85,B 0,C 180,E1 -21608.078,E2 -21608.078} C_VEL
LIN {X 0,Y 199.841,Z 325.578,A -85,B 0,C 180,E1 -21612.181,E2 -21612.181} C_VEL
LIN {X 0,Y 199.763,Z 325.586,A -85,B 0,C 180,E1 -21616.347,E2 -21616.347} C_VEL
LIN {X 0,Y 199.716,Z 325.591,A -85,B 0,C 180,E1 -21620.604,E2 -21620.604} C_VEL
LIN {X 0,Y 199.646,Z 325.601,A -85,B 0,C 180,E1 -21624.988,E2 -21624.988} C_VEL
LIN {X 0,Y 199.641,Z 325.61,A -85,B 0,C 180,E1 -21629.528,E2 -21629.528} C_VEL
LIN {X 0,Y 199.67,Z 325.767,A -85,B 0,C 180,E1 -21630.982,E2 -21630.982} C_VEL
LIN {X 0,Y 201.075,Z 329.678,A -85,B 0,C 180,E1 -21635.274,E2 -21635.274} C_VEL
LIN {X 0,Y 204.211,Z 334.17,A -85,B 0,C 180,E1 -21637.545,E2 -21637.545} C_VEL
LIN {X 0,Y 206.487,Z 336.944,A -85,B 0,C 180,E1 -21638.99,E2 -21638.99} C_VEL
LIN {X 0,Y 210.148,Z 342.207,A -85,B 0,C 180,E1 -21641.174,E2 -21641.174} C_VEL
LIN {X 0,Y 215.093,Z 350.015,A -85,B 0,C 180,E1 -21643.773,E2 -21643.773} C_VEL
LIN {X 0,Y 218.099,Z 355.037,A -85,B 0,C 180,E1 -21645.218,E2 -21645.218} C_VEL
LIN {X 0,Y 218.238,Z 355.296,A -85,B 0,C 180,E1 -21645.285,E2 -21645.285} C_VEL
LIN {X 0,Y 220.088,Z 359.672,A -85,B 0,C 180,E1 -21646.199,E2 -21646.199} C_VEL
LIN {X 0,Y 221.45,Z 364.685,A -85,B 0,C 180,E1 -21646.946,E2 -21646.946} C_VEL
LIN {X 0,Y 223.556,Z 375.445,A -85,B 0,C 180,E1 -21648.218,E2 -21648.218} C_VEL
LIN {X 0,Y 225.344,Z 382.395,A -85,B 0,C 180,E1 -21649.138,E2 -21649.138} C_VEL
LIN {X 0,Y 227.47,Z 388.187,A -85,B 0,C 180,E1 -21650.043,E2 -21650.043} C_VEL
LIN {X 0,Y 228.154,Z 396.647,A -85,B 0,C 180,E1 -21650.661,E2 -21650.661} C_VEL
LIN {X 0,Y 224.94,Z 441.599,A -85,B 0,C 180,E1 -21652.152,E2 -21652.152} C_VEL
LIN {X 0,Y 223.066,Z 455.256,A -85,B 0,C 180,E1 -21652.904,E2 -21652.904} C_VEL
LIN {X 0,Y 220.506,Z 467.669,A -85,B 0,C 180,E1 -21653.879,E2 -21653.879} C_VEL
LIN {X 0,Y 217.288,Z 480.041,A -85,B 0,C 180,E1 -21655.255,E2 -21655.255} C_VEL
LIN {X 0,Y 213.864,Z 491.153,A -85,B 0,C 180,E1 -21656.894,E2 -21656.894} C_VEL
LIN {X 0,Y 210.23,Z 501.273,A -85,B 0,C 180,E1 -21658.8,E2 -21658.8} C_VEL
LIN {X 0,Y 206.563,Z 510.459,A -85,B 0,C 180,E1 -21661.008,E2 -21661.008} C_VEL
LIN {X 0,Y 202.612,Z 519.441,A -85,B 0,C 180,E1 -21663.761,E2 -21663.761} C_VEL
LIN {X 0,Y 199.319,Z 526.764,A -85,B 0,C 180,E1 -21666.663,E2 -21666.663} C_VEL
LIN {X 0,Y 196.837,Z 531.67,A -85,B 0,C 180,E1 -21669.09,E2 -21669.09} C_VEL
LIN {X 0,Y 194.422,Z 536.521,A -85,B 0,C 180,E1 -21672.114,E2 -21672.114} C_VEL
LIN {X 0,Y 192.491,Z 540.281,A -85,B 0,C 180,E1 -21675.2,E2 -21675.2} C_VEL
LIN {X 0,Y 191.644,Z 542.249,A -85,B 0,C 180,E1 -21677.297,E2 -21677.297} C_VEL
LIN {X 0,Y 190.984,Z 543.795,A -85,B 0,C 180,E1 -21679.405,E2 -21679.405} C_VEL
LIN {X 0,Y 190.273,Z 545.631,A -85,B 0,C 180,E1 -21683.645,E2 -21683.645} C_VEL
LIN {X 0,Y 190.152,Z 546.002,A -85,B 0,C 180,E1 -21686.302,E2 -21686.302} C_VEL
LIN {X 0,Y 190.405,Z 545.43,A -85,B 0,C 180,E1 -21690.007,E2 -21690.007} C_VEL
LIN {X 0,Y 190.279,Z 544.52,A -85,B 0,C 180,E1 -21692.123,E2 -21692.123} C_VEL
LIN {X 0,Y 190.246,Z 543.201,A -85,B 0,C 180,E1 -21694.244,E2 -21694.244} C_VEL
LIN {X 0,Y 190.417,Z 540.365,A -85,B 0,C 180,E1 -21697.429,E2 -21697.429} C_VEL
LIN {X 0,Y 190.935,Z 536.458,A -85,B 0,C 180,E1 -21700.611,E2 -21700.611} C_VEL
LIN {X 0,Y 192.061,Z 530.4,A -85,B 0,C 180,E1 -21704.306,E2 -21704.306} C_VEL
LIN {X 0,Y 193.697,Z 523.72,A -85,B 0,C 180,E1 -21707.424,E2 -21707.424} C_VEL
LIN {X 0,Y 195.43,Z 516.907,A -85,B 0,C 180,E1 -21709.982,E2 -21709.982} C_VEL
LIN {X 0,Y 196.94,Z 510.467,A -85,B 0,C 180,E1 -21712.01,E2 -21712.01} C_VEL
LIN {X 0,Y 199.245,Z 500.763,A -85,B 0,C 180,E1 -21714.491,E2 -21714.491} C_VEL
LIN {X 0,Y 201.695,Z 490.022,A -85,B 0,C 180,E1 -21716.661,E2 -21716.661} C_VEL
LIN {X 0,Y 203.908,Z 479.687,A -85,B 0,C 180,E1 -21718.294,E2 -21718.294} C_VEL
LIN {X 0,Y 205.863,Z 468.466,A -85,B 0,C 180,E1 -21719.676,E2 -21719.676} C_VEL
LIN {X 0,Y 207.63,Z 455.232,A -85,B 0,C 180,E1 -21720.87,E2 -21720.87} C_VEL
LIN {X 0,Y 208.89,Z 442.306,A -85,B 0,C 180,E1 -21721.649,E2 -21721.649} C_VEL
LIN {X 0,Y 211.347,Z 392.58,A -85,B 0,C 180,E1 -21723.418,E2 -21723.418} C_VEL
LIN {X 0,Y 208.588,Z 368.774,A -85,B 0,C 180,E1 -21724.803,E2 -21724.803} C_VEL
LIN {X 0,Y 200.937,Z 348.809,A -85,B 0,C 180,E1 -21726.862,E2 -21726.862} C_VEL
LIN {X 0,Y 194.289,Z 333.55,A -85,B 0,C 180,E1 -21728.765,E2 -21728.765} C_VEL
LIN {X 0,Y 192.52,Z 326.502,A -85,B 0,C 180,E1 -21732.618,E2 -21732.618} C_VEL
LIN {X 0,Y 192.497,Z 326.511,A -85,B 0,C 180,E1 -21736.908,E2 -21736.908} C_VEL
LIN {X 0,Y 192.551,Z 326.5,A -85,B 0,C 180,E1 -21741.648,E2 -21741.648} C_VEL
LIN {X 0,Y 192.606,Z 326.497,A -85,B 0,C 180,E1 -21746.816,E2 -21746.816} C_VEL
LIN {X 0,Y 192.67,Z 326.486,A -85,B 0,C 180,E1 -21751.693,E2 -21751.693} C_VEL
LIN {X 0,Y 192.682,Z 326.481,A -85,B 0,C 180,E1 -21756.345,E2 -21756.345} C_VEL
LIN {X 0,Y 192.704,Z 326.463,A -85,B 0,C 180,E1 -21761.493,E2 -21761.493} C_VEL
LIN {X 0,Y 192.74,Z 326.45,A -85,B 0,C 180,E1 -21765.212,E2 -21765.212} C_VEL
LIN {X 0,Y 192.955,Z 326.45,A -85,B 0,C 180,E1 -21769.567,E2 -21769.567} C_VEL
LIN {X 0,Y 192.984,Z 326.433,A -85,B 0,C 180,E1 -21773.728,E2 -21773.728} C_VEL
LIN {X 0,Y 193.251,Z 326.368,A -85,B 0,C 180,E1 -21777.916,E2 -21777.916} C_VEL
LIN {X 0,Y 193.438,Z 326.358,A -85,B 0,C 180,E1 -21780,E2 -21780} C_VEL
LIN {X 0,Y 192.959,Z 326.447,A -85,B 0,C 180,E1 -21784.177,E2 -21784.177} C_VEL
LIN {X 0,Y 193.025,Z 326.435,A -85,B 0,C 180,E1 -21788.374,E2 -21788.374} C_VEL
LIN {X 0,Y 192.792,Z 326.466,A -85,B 0,C 180,E1 -21792.634,E2 -21792.634} C_VEL
LIN {X 0,Y 192.716,Z 326.474,A -85,B 0,C 180,E1 -21796.963,E2 -21796.963} C_VEL
LIN {X 0,Y 192.584,Z 326.491,A -85,B 0,C 180,E1 -21801.404,E2 -21801.404} C_VEL
LIN {X 0,Y 192.626,Z 326.488,A -85,B 0,C 180,E1 -21804.191,E2 -21804.191} C_VEL
LIN {X 0,Y 192.594,Z 326.468,A -85,B 0,C 180,E1 -21808.855,E2 -21808.855} C_VEL
LIN {X 0,Y 192.571,Z 326.463,A -85,B 0,C 180,E1 -21813.191,E2 -21813.191} C_VEL
LIN {X 0,Y 192.589,Z 326.488,A -85,B 0,C 180,E1 -21816.593,E2 -21816.593} C_VEL
LIN {X 0,Y 192.511,Z 326.5,A -85,B 0,C 180,E1 -21821.081,E2 -21821.081} C_VEL
LIN {X 0,Y 192.494,Z 326.507,A -85,B 0,C 180,E1 -21826.071,E2 -21826.071} C_VEL
LIN {X 0,Y 192.512,Z 326.497,A -85,B 0,C 180,E1 -21830.054,E2 -21830.054} C_VEL
LIN {X 0,Y 192.566,Z 326.498,A -85,B 0,C 180,E1 -21834.266,E2 -21834.266} C_VEL
LIN {X 0,Y 192.612,Z 326.493,A -85,B 0,C 180,E1 -21837.058,E2 -21837.058} C_VEL
LIN {X 0,Y 192.625,Z 326.49,A -85,B 0,C 180,E1 -21841.68,E2 -21841.68} C_VEL
LIN {X 0,Y 192.679,Z 326.483,A -85,B 0,C 180,E1 -21846.339,E2 -21846.339} C_VEL
LIN {X 0,Y 192.702,Z 326.484,A -85,B 0,C 180,E1 -21851.486,E2 -21851.486} C_VEL
LIN {X 0,Y 192.744,Z 326.476,A -85,B 0,C 180,E1 -21855.206,E2 -21855.206} C_VEL
LIN {X 0,Y 192.951,Z 326.451,A -85,B 0,C 180,E1 -21859.561,E2 -21859.561} C_VEL
LIN {X 0,Y 192.996,Z 326.582,A -85,B 0,C 180,E1 -21863.394,E2 -21863.394} C_VEL
LIN {X 0,Y 194.001,Z 329.355,A -85,B 0,C 180,E1 -21863.709,E2 -21863.709} C_VEL
LIN {X 0,Y 203.085,Z 345.732,A -85,B 0,C 180,E1 -21866.004,E2 -21866.004} C_VEL
LIN {X 0,Y 206.396,Z 353.14,A -85,B 0,C 180,E1 -21866.852,E2 -21866.852} C_VEL
LIN {X 0,Y 212.257,Z 368.813,A -85,B 0,C 180,E1 -21868.379,E2 -21868.379} C_VEL
LIN {X 0,Y 209.221,Z 428.247,A -85,B 0,C 180,E1 -21870.475,E2 -21870.475} C_VEL
LIN {X 0,Y 208.044,Z 441.746,A -85,B 0,C 180,E1 -21871.324,E2 -21871.324} C_VEL
LIN {X 0,Y 206.426,Z 454.887,A -85,B 0,C 180,E1 -21872.555,E2 -21872.555} C_VEL
LIN {X 0,Y 204.352,Z 467.333,A -85,B 0,C 180,E1 -21874.161,E2 -21874.161} C_VEL
LIN {X 0,Y 202.162,Z 478.225,A -85,B 0,C 180,E1 -21875.979,E2 -21875.979} C_VEL
LIN {X 0,Y 199.921,Z 488.179,A -85,B 0,C 180,E1 -21878.076,E2 -21878.076} C_VEL
LIN {X 0,Y 197.554,Z 498.168,A -85,B 0,C 180,E1 -21880.757,E2 -21880.757} C_VEL
LIN {X 0,Y 195.33,Z 506.936,A -85,B 0,C 180,E1 -21883.72,E2 -21883.72} C_VEL
LIN {X 0,Y 193.514,Z 514.266,A -85,B 0,C 180,E1 -21886.882,E2 -21886.882} C_VEL
LIN {X 0,Y 192.015,Z 520.474,A -85,B 0,C 180,E1 -21890.339,E2 -21890.339} C_VEL
LIN {X 0,Y 191.03,Z 525.264,A -85,B 0,C 180,E1 -21893.862,E2 -21893.862} C_VEL
LIN {X 0,Y 190.185,Z 528.811,A -85,B 0,C 180,E1 -21897.515,E2 -21897.515} C_VEL
LIN {X 0,Y 189.875,Z 531.217,A -85,B 0,C 180,E1 -21901.644,E2 -21901.644} C_VEL
LIN {X 0,Y 190.142,Z 532.119,A -85,B 0,C 180,E1 -21905.594,E2 -21905.594} C_VEL
LIN {X 0,Y 190.917,Z 531.687,A -85,B 0,C 180,E1 -21909.371,E2 -21909.371} C_VEL
LIN {X 0,Y 192.209,Z 530.032,A -85,B 0,C 180,E1 -21913.005,E2 -21913.005} C_VEL
LIN {X 0,Y 193.946,Z 527.264,A -85,B 0,C 180,E1 -21916.488,E2 -21916.488} C_VEL
LIN {X 0,Y 196.177,Z 523.353,A -85,B 0,C 180,E1 -21919.846,E2 -21919.846} C_VEL
LIN {X 0,Y 199.002,Z 518.157,A -85,B 0,C 180,E1 -21923.103,E2 -21923.103} C_VEL
LIN {X 0,Y 202.547,Z 511.22,A -85,B 0,C 180,E1 -21926.365,E2 -21926.365} C_VEL
LIN {X 0,Y 206.366,Z 503.033,A -85,B 0,C 180,E1 -21929.28,E2 -21929.28} C_VEL
LIN {X 0,Y 210.169,Z 493.822,A -85,B 0,C 180,E1 -21931.853,E2 -21931.853} C_VEL
LIN {X 0,Y 213.467,Z 485.089,A -85,B 0,C 180,E1 -21933.765,E2 -21933.765} C_VEL
LIN {X 0,Y 216.966,Z 474.339,A -85,B 0,C 180,E1 -21935.625,E2 -21935.625} C_VEL
LIN {X 0,Y 220.114,Z 462.705,A -85,B 0,C 180,E1 -21937.187,E2 -21937.187} C_VEL
LIN {X 0,Y 222.617,Z 451.149,A -85,B 0,C 180,E1 -21938.367,E2 -21938.367} C_VEL
LIN {X 0,Y 224.55,Z 438.505,A -85,B 0,C 180,E1 -21939.317,E2 -21939.317} C_VEL
LIN {X 0,Y 226.035,Z 425.433,A -85,B 0,C 180,E1 -21939.912,E2 -21939.912} C_VEL
LIN {X 0,Y 229.002,Z 381.421,A -85,B 0,C 180,E1 -21941.362,E2 -21941.362} C_VEL
LIN {X 0,Y 224.799,Z 372.022,A -85,B 0,C 180,E1 -21943.074,E2 -21943.074} C_VEL
LIN {X 0,Y 219.89,Z 363.192,A -85,B 0,C 180,E1 -21945.138,E2 -21945.138} C_VEL
LIN {X 0,Y 214.175,Z 354.431,A -85,B 0,C 180,E1 -21947.776,E2 -21947.776} C_VEL
LIN {X 0,Y 212.044,Z 351.389,A -85,B 0,C 180,E1 -21948.833,E2 -21948.833} C_VEL
LIN {X 0,Y 208.914,Z 347.041,A -85,B 0,C 180,E1 -21950.517,E2 -21950.517} C_VEL
LIN {X 0,Y 206.287,Z 343.214,A -85,B 0,C 180,E1 -21952.077,E2 -21952.077} C_VEL
LIN {X 0,Y 203.342,Z 339.821,A -85,B 0,C 180,E1 -21953.914,E2 -21953.914} C_VEL
LIN {X 0,Y 202.163,Z 337.837,A -85,B 0,C 180,E1 -21954.764,E2 -21954.764} C_VEL
LIN {X 0,Y 199.589,Z 335.626,A -85,B 0,C 180,E1 -21956.593,E2 -21956.593} C_VEL
LIN {X 0,Y 198.156,Z 332.816,A -85,B 0,C 180,E1 -21957.904,E2 -21957.904} C_VEL
LIN {X 0,Y 197.823,Z 332.192,A -85,B 0,C 180,E1 -21958.219,E2 -21958.219} C_VEL
LIN {X 0,Y 194.818,Z 329.976,A -85,B 0,C 180,E1 -21960.904,E2 -21960.904} C_VEL
LIN {X 0,Y 193.178,Z 327.013,A -85,B 0,C 180,E1 -21962.933,E2 -21962.933} C_VEL
LIN {X 0,Y 193.035,Z 326.427,A -85,B 0,C 180,E1 -21963.261,E2 -21963.261} C_VEL
LIN {X 0,Y 193.008,Z 326.431,A -85,B 0,C 180,E1 -21968.375,E2 -21968.375} C_VEL
LIN {X 0,Y 192.767,Z 326.46,A -85,B 0,C 180,E1 -21972.636,E2 -21972.636} C_VEL
LIN {X 0,Y 192.732,Z 326.463,A -85,B 0,C 180,E1 -21976.961,E2 -21976.961} C_VEL
LIN {X 0,Y 192.641,Z 326.475,A -85,B 0,C 180,E1 -21981.397,E2 -21981.397} C_VEL
LIN {X 0,Y 192.59,Z 326.483,A -85,B 0,C 180,E1 -21985.48,E2 -21985.48} C_VEL
LIN {X 0,Y 193.305,Z 328.733,A -85,B 0,C 180,E1 -21988.96,E2 -21988.96} C_VEL
LIN {X 0,Y 198.144,Z 335.011,A -85,B 0,C 180,E1 -21993.809,E2 -21993.809} C_VEL
LIN {X 0,Y 199.238,Z 336.441,A -85,B 0,C 180,E1 -21994.734,E2 -21994.734} C_VEL
LIN {X 0,Y 204.15,Z 343.237,A -85,B 0,C 180,E1 -21998.292,E2 -21998.292} C_VEL
LIN {X 0,Y 208.194,Z 349.34,A -85,B 0,C 180,E1 -22000.805,E2 -22000.805} C_VEL
LIN {X 0,Y 212.503,Z 356.4,A -85,B 0,C 180,E1 -22003.172,E2 -22003.172} C_VEL
LIN {X 0,Y 215.198,Z 361.152,A -85,B 0,C 180,E1 -22004.536,E2 -22004.536} C_VEL
LIN {X 0,Y 219.896,Z 369.989,A -85,B 0,C 180,E1 -22006.742,E2 -22006.742} C_VEL
LIN {X 0,Y 224.789,Z 380.874,A -85,B 0,C 180,E1 -22008.89,E2 -22008.89} C_VEL
LIN {X 0,Y 225.344,Z 382.395,A -85,B 0,C 180,E1 -22009.138,E2 -22009.138} C_VEL
LIN {X 0,Y 226.07,Z 385.911,A -85,B 0,C 180,E1 -22009.535,E2 -22009.535} C_VEL
LIN {X 0,Y 226.04,Z 391.738,A -85,B 0,C 180,E1 -22009.831,E2 -22009.831} C_VEL
LIN {X 0,Y 225.128,Z 397.712,A -85,B 0,C 180,E1 -22009.888,E2 -22009.888} C_VEL
LIN {X 0,Y 222.62,Z 409.927,A -85,B 0,C 180,E1 -22009.821,E2 -22009.821} C_VEL
LIN {X 0,Y 222.151,Z 414.024,A -85,B 0,C 180,E1 -22009.907,E2 -22009.907} C_VEL
LIN {X 0,Y 219.978,Z 441.699,A -85,B 0,C 180,E1 -22010.843,E2 -22010.843} C_VEL
LIN {X 0,Y 218.005,Z 455.246,A -85,B 0,C 180,E1 -22011.594,E2 -22011.594} C_VEL
LIN {X 0,Y 215.38,Z 467.583,A -85,B 0,C 180,E1 -22012.584,E2 -22012.584} C_VEL
LIN {X 0,Y 212.028,Z 479.915,A -85,B 0,C 180,E1 -22013.97,E2 -22013.97} C_VEL
LIN {X 0,Y 208.447,Z 491.004,A -85,B 0,C 180,E1 -22015.626,E2 -22015.626} C_VEL
LIN {X 0,Y 204.646,Z 501.098,A -85,B 0,C 180,E1 -22017.558,E2 -22017.558} C_VEL
LIN {X 0,Y 200.415,Z 511.045,A -85,B 0,C 180,E1 -22020.029,E2 -22020.029} C_VEL
LIN {X 0,Y 196.291,Z 519.855,A -85,B 0,C 180,E1 -22022.848,E2 -22022.848} C_VEL
LIN {X 0,Y 193.191,Z 526.175,A -85,B 0,C 180,E1 -22025.432,E2 -22025.432} C_VEL
LIN {X 0,Y 190.212,Z 531.852,A -85,B 0,C 180,E1 -22028.325,E2 -22028.325} C_VEL
LIN {X 0,Y 187.667,Z 536.608,A -85,B 0,C 180,E1 -22031.447,E2 -22031.447} C_VEL
LIN {X 0,Y 185.603,Z 540.278,A -85,B 0,C 180,E1 -22034.638,E2 -22034.638} C_VEL
LIN {X 0,Y 184.702,Z 542.197,A -85,B 0,C 180,E1 -22036.811,E2 -22036.811} C_VEL
LIN {X 0,Y 183.492,Z 544.731,A -85,B 0,C 180,E1 -22041.195,E2 -22041.195} C_VEL
LIN {X 0,Y 183.076,Z 545.722,A -85,B 0,C 180,E1 -22045.604,E2 -22045.604} C_VEL
LIN {X 0,Y 183.141,Z 545.601,A -85,B 0,C 180,E1 -22047.808,E2 -22047.808} C_VEL
LIN {X 0,Y 183.322,Z 545.072,A -85,B 0,C 180,E1 -22050.007,E2 -22050.007} C_VEL
LIN {X 0,Y 183.157,Z 543.089,A -85,B 0,C 180,E1 -22053.919,E2 -22053.919} C_VEL
LIN {X 0,Y 183.352,Z 539.851,A -85,B 0,C 180,E1 -22057.717,E2 -22057.717} C_VEL
LIN {X 0,Y 183.916,Z 535.859,A -85,B 0,C 180,E1 -22061.021,E2 -22061.021} C_VEL
LIN {X 0,Y 185.153,Z 529.663,A -85,B 0,C 180,E1 -22064.852,E2 -22064.852} C_VEL
LIN {X 0,Y 186.85,Z 522.872,A -85,B 0,C 180,E1 -22068.084,E2 -22068.084} C_VEL
LIN {X 0,Y 188.885,Z 514.834,A -85,B 0,C 180,E1 -22071.118,E2 -22071.118} C_VEL
LIN {X 0,Y 191.257,Z 505.67,A -85,B 0,C 180,E1 -22073.847,E2 -22073.847} C_VEL
LIN {X 0,Y 193.649,Z 496.101,A -85,B 0,C 180,E1 -22076.112,E2 -22076.112} C_VEL
LIN {X 0,Y 195.938,Z 485.657,A -85,B 0,C 180,E1 -22078.09,E2 -22078.09} C_VEL
LIN {X 0,Y 197.897,Z 476.034,A -85,B 0,C 180,E1 -22079.527,E2 -22079.527} C_VEL
LIN {X 0,Y 199.987,Z 463.854,A -85,B 0,C 180,E1 -22080.933,E2 -22080.933} C_VEL
LIN {X 0,Y 201.74,Z 450.332,A -85,B 0,C 180,E1 -22082.022,E2 -22082.022} C_VEL
LIN {X 0,Y 202.866,Z 436.961,A -85,B 0,C 180,E1 -22082.704,E2 -22082.704} C_VEL
LIN {X 0,Y 204.908,Z 392.318,A -85,B 0,C 180,E1 -22084.332,E2 -22084.332} C_VEL
LIN {X 0,Y 202.361,Z 370.69,A -85,B 0,C 180,E1 -22085.661,E2 -22085.661} C_VEL
LIN {X 0,Y 195.113,Z 351.772,A -85,B 0,C 180,E1 -22087.706,E2 -22087.706} C_VEL
LIN {X 0,Y 188.592,Z 337.026,A -85,B 0,C 180,E1 -22089.589,E2 -22089.589} C_VEL
LIN {X 0,Y 187.009,Z 333.359,A -85,B 0,C 180,E1 -22090.083,E2 -22090.083} C_VEL
LIN {X 0,Y 185.459,Z 327.383,A -85,B 0,C 180,E1 -22093.57,E2 -22093.57} C_VEL
LIN {X 0,Y 185.464,Z 327.387,A -85,B 0,C 180,E1 -22096.992,E2 -22096.992} C_VEL
LIN {X 0,Y 185.467,Z 327.382,A -85,B 0,C 180,E1 -22099.895,E2 -22099.895} C_VEL
LIN {X 0,Y 185.51,Z 327.379,A -85,B 0,C 180,E1 -22102.716,E2 -22102.716} C_VEL
LIN {X 0,Y 185.551,Z 327.374,A -85,B 0,C 180,E1 -22107.976,E2 -22107.976} C_VEL
LIN {X 0,Y 185.591,Z 327.365,A -85,B 0,C 180,E1 -22110.579,E2 -22110.579} C_VEL
LIN {X 0,Y 185.591,Z 327.362,A -85,B 0,C 180,E1 -22115.383,E2 -22115.383} C_VEL
LIN {X 0,Y 185.635,Z 327.344,A -85,B 0,C 180,E1 -22121.18,E2 -22121.18} C_VEL
LIN {X 0,Y 185.67,Z 327.326,A -85,B 0,C 180,E1 -22124.635,E2 -22124.635} C_VEL
LIN {X 0,Y 185.898,Z 327.329,A -85,B 0,C 180,E1 -22129.42,E2 -22129.42} C_VEL
LIN {X 0,Y 185.947,Z 327.31,A -85,B 0,C 180,E1 -22133.489,E2 -22133.489} C_VEL
LIN {X 0,Y 186.197,Z 327.245,A -85,B 0,C 180,E1 -22137.837,E2 -22137.837} C_VEL
LIN {X 0,Y 186.403,Z 327.232,A -85,B 0,C 180,E1 -22140,E2 -22140} C_VEL
LIN {X 0,Y 185.906,Z 327.325,A -85,B 0,C 180,E1 -22144.336,E2 -22144.336} C_VEL
LIN {X 0,Y 185.977,Z 327.312,A -85,B 0,C 180,E1 -22148.694,E2 -22148.694} C_VEL
LIN {X 0,Y 185.717,Z 327.347,A -85,B 0,C 180,E1 -22153.124,E2 -22153.124} C_VEL
LIN {X 0,Y 185.635,Z 327.346,A -85,B 0,C 180,E1 -22158.819,E2 -22158.819} C_VEL
LIN {X 0,Y 185.555,Z 327.367,A -85,B 0,C 180,E1 -22164.622,E2 -22164.622} C_VEL
LIN {X 0,Y 185.509,Z 327.339,A -85,B 0,C 180,E1 -22169.506,E2 -22169.506} C_VEL
LIN {X 0,Y 185.494,Z 327.357,A -85,B 0,C 180,E1 -22174.633,E2 -22174.633} C_VEL
LIN {X 0,Y 185.509,Z 327.373,A -85,B 0,C 180,E1 -22177.312,E2 -22177.312} C_VEL
LIN {X 0,Y 185.469,Z 327.379,A -85,B 0,C 180,E1 -22180.718,E2 -22180.718} C_VEL
LIN {X 0,Y 185.463,Z 327.382,A -85,B 0,C 180,E1 -22186.054,E2 -22186.054} C_VEL
LIN {X 0,Y 185.463,Z 327.375,A -85,B 0,C 180,E1 -22189.888,E2 -22189.888} C_VEL
LIN {X 0,Y 185.51,Z 327.38,A -85,B 0,C 180,E1 -22192.711,E2 -22192.711} C_VEL
LIN {X 0,Y 185.537,Z 327.376,A -85,B 0,C 180,E1 -22197.968,E2 -22197.968} C_VEL
LIN {X 0,Y 185.555,Z 327.371,A -85,B 0,C 180,E1 -22200.592,E2 -22200.592} C_VEL
LIN {X 0,Y 185.589,Z 327.367,A -85,B 0,C 180,E1 -22205.377,E2 -22205.377} C_VEL
LIN {X 0,Y 185.633,Z 327.363,A -85,B 0,C 180,E1 -22211.173,E2 -22211.173} C_VEL
LIN {X 0,Y 185.673,Z 327.355,A -85,B 0,C 180,E1 -22214.629,E2 -22214.629} C_VEL
LIN {X 0,Y 185.893,Z 327.331,A -85,B 0,C 180,E1 -22219.413,E2 -22219.413} C_VEL
LIN {X 0,Y 185.992,Z 327.31,A -85,B 0,C 180,E1 -22222.053,E2 -22222.053} C_VEL
LIN {X 0,Y 187.008,Z 330.226,A -85,B 0,C 180,E1 -22222.436,E2 -22222.436} C_VEL
LIN {X 0,Y 197.576,Z 349.425,A -85,B 0,C 180,E1 -22225.267,E2 -22225.267} C_VEL
LIN {X 0,Y 200.928,Z 357.025,A -85,B 0,C 180,E1 -22226.156,E2 -22226.156} C_VEL
LIN {X 0,Y 205.896,Z 370.453,A -85,B 0,C 180,E1 -22227.521,E2 -22227.521} C_VEL
LIN {X 0,Y 202.804,Z 428.715,A -85,B 0,C 180,E1 -22229.638,E2 -22229.638} C_VEL
LIN {X 0,Y 201.528,Z 442.704,A -85,B 0,C 180,E1 -22230.555,E2 -22230.555} C_VEL
LIN {X 0,Y 199.928,Z 455.084,A -85,B 0,C 180,E1 -22231.756,E2 -22231.756} C_VEL
LIN {X 0,Y 197.929,Z 466.833,A -85,B 0,C 180,E1 -22233.301,E2 -22233.301} C_VEL
LIN {X 0,Y 195.37,Z 479.14,A -85,B 0,C 180,E1 -22235.411,E2 -22235.411} C_VEL
LIN {X 0,Y 192.795,Z 490.017,A -85,B 0,C 180,E1 -22237.85,E2 -22237.85} C_VEL
LIN {X 0,Y 190.373,Z 499.756,A -85,B 0,C 180,E1 -22240.629,E2 -22240.629} C_VEL
LIN {X 0,Y 188.124,Z 508.367,A -85,B 0,C 180,E1 -22243.755,E2 -22243.755} C_VEL
LIN {X 0,Y 186.276,Z 515.372,A -85,B 0,C 180,E1 -22246.993,E2 -22246.993} C_VEL
LIN {X 0,Y 185.009,Z 520.505,A -85,B 0,C 180,E1 -22249.983,E2 -22249.983} C_VEL
LIN {X 0,Y 183.991,Z 525.241,A -85,B 0,C 180,E1 -22253.546,E2 -22253.546} C_VEL
LIN {X 0,Y 183.094,Z 528.95,A -85,B 0,C 180,E1 -22257.417,E2 -22257.417} C_VEL
LIN {X 0,Y 182.829,Z 530.602,A -85,B 0,C 180,E1 -22259.971,E2 -22259.971} C_VEL
LIN {X 0,Y 182.807,Z 531.748,A -85,B 0,C 180,E1 -22262.552,E2 -22262.552} C_VEL
LIN {X 0,Y 183.16,Z 532.416,A -85,B 0,C 180,E1 -22266.313,E2 -22266.313} C_VEL
LIN {X 0,Y 184.126,Z 531.787,A -85,B 0,C 180,E1 -22270.444,E2 -22270.444} C_VEL
LIN {X 0,Y 185.467,Z 530.149,A -85,B 0,C 180,E1 -22273.947,E2 -22273.947} C_VEL
LIN {X 0,Y 187.401,Z 527.306,A -85,B 0,C 180,E1 -22277.542,E2 -22277.542} C_VEL
LIN {X 0,Y 189.861,Z 523.307,A -85,B 0,C 180,E1 -22281.003,E2 -22281.003} C_VEL
LIN {X 0,Y 192.961,Z 517.997,A -85,B 0,C 180,E1 -22284.355,E2 -22284.355} C_VEL
LIN {X 0,Y 196.609,Z 511.216,A -85,B 0,C 180,E1 -22287.575,E2 -22287.575} C_VEL
